LIN {X 0,Y 256.306,Z 543.369,A -85,B 0,C 180,E1 -18708.933,E2 -18708.933} C_VEL
LIN {X 0,Y 256.535,Z 543.34,A -85,B 0,C 180,E1 -18712.126,E2 -18712.126} C_VEL
LIN {X 0,Y 256.709,Z 543.322,A -85,B 0,C 180,E1 -18718.431,E2 -18718.431} C_VEL
LIN {X 0,Y 256.709,Z 543.317,A -85,B 0,C 180,E1 -18721.568,E2 -18721.568} C_VEL
LIN {X 0,Y 256.532,Z 543.34,A -85,B 0,C 180,E1 -18727.873,E2 -18727.873} C_VEL
LIN {X 0,Y 256.304,Z 543.369,A -85,B 0,C 180,E1 -18731.066,E2 -18731.066} C_VEL
LIN {X 0,Y 256.289,Z 543.37,A -85,B 0,C 180,E1 -18735.915,E2 -18735.915} C_VEL
LIN {X 0,Y 256.155,Z 543.39,A -85,B 0,C 180,E1 -18740.925,E2 -18740.925} C_VEL
LIN {X 0,Y 256.166,Z 543.386,A -85,B 0,C 180,E1 -18745.13,E2 -18745.13} C_VEL
LIN {X 0,Y 256.134,Z 543.388,A -85,B 0,C 180,E1 -18747.754,E2 -18747.754} C_VEL
LIN {X 0,Y 255.867,Z 543.426,A -85,B 0,C 180,E1 -18748.632,E2 -18748.632} C_VEL
LIN {X 0,Y 254.547,Z 543.595,A -85,B 0,C 180,E1 -18749.928,E2 -18749.928} C_VEL
LIN {X 0,Y 250.177,Z 544.136,A -85,B 0,C 180,E1 -18752.946,E2 -18752.946} C_VEL
LIN {X 0,Y 249.117,Z 544.265,A -85,B 0,C 180,E1 -18754.298,E2 -18754.298} C_VEL
LIN {X 0,Y 249.035,Z 544.274,A -85,B 0,C 180,E1 -18754.757,E2 -18754.757} C_VEL
LIN {X 0,Y 249.021,Z 544.276,A -85,B 0,C 180,E1 -18758.381,E2 -18758.381} C_VEL
LIN {X 0,Y 249.008,Z 544.281,A -85,B 0,C 180,E1 -18762.793,E2 -18762.793} C_VEL
LIN {X 0,Y 249.015,Z 544.278,A -85,B 0,C 180,E1 -18767.364,E2 -18767.364} C_VEL
LIN {X 0,Y 249.084,Z 544.269,A -85,B 0,C 180,E1 -18772.188,E2 -18772.188} C_VEL
LIN {X 0,Y 249.237,Z 544.478,A -85,B 0,C 180,E1 -18773.377,E2 -18773.377} C_VEL
LIN {X 0,Y 251.469,Z 555.944,A -85,B 0,C 180,E1 -18777.927,E2 -18777.927} C_VEL
LIN {X 0,Y 252.35,Z 561.158,A -85,B 0,C 180,E1 -18779.914,E2 -18779.914} C_VEL
LIN {X 0,Y 250.485,Z 573.384,A -85,B 0,C 180,E1 -18784.422,E2 -18784.422} C_VEL
LIN {X 0,Y 249.648,Z 580.162,A -85,B 0,C 180,E1 -18786.831,E2 -18786.831} C_VEL
LIN {X 0,Y 249.979,Z 590.6,A -85,B 0,C 180,E1 -18787.367,E2 -18787.367} C_VEL
LIN {X 0,Y 253.841,Z 654.438,A -85,B 0,C 180,E1 -18790.307,E2 -18790.307} C_VEL
LIN {X 0,Y 253.269,Z 669.393,A -85,B 0,C 180,E1 -18791.024,E2 -18791.024} C_VEL
LIN {X 0,Y 252.559,Z 681.968,A -85,B 0,C 180,E1 -18791.967,E2 -18791.967} C_VEL
LIN {X 0,Y 251.556,Z 693.327,A -85,B 0,C 180,E1 -18793.151,E2 -18793.151} C_VEL
LIN {X 0,Y 250.486,Z 703.576,A -85,B 0,C 180,E1 -18794.541,E2 -18794.541} C_VEL
LIN {X 0,Y 249.573,Z 714,A -85,B 0,C 180,E1 -18796.359,E2 -18796.359} C_VEL
LIN {X 0,Y 248.841,Z 722.24,A -85,B 0,C 180,E1 -18798.185,E2 -18798.185} C_VEL
LIN {X 0,Y 248.424,Z 729.674,A -85,B 0,C 180,E1 -18800.227,E2 -18800.227} C_VEL
LIN {X 0,Y 248.37,Z 736.358,A -85,B 0,C 180,E1 -18802.588,E2 -18802.588} C_VEL
LIN {X 0,Y 248.68,Z 741.797,A -85,B 0,C 180,E1 -18805.136,E2 -18805.136} C_VEL
LIN {X 0,Y 248.915,Z 744.383,A -85,B 0,C 180,E1 -18806.763,E2 -18806.763} C_VEL
LIN {X 0,Y 249.202,Z 746.318,A -85,B 0,C 180,E1 -18808.384,E2 -18808.384} C_VEL
LIN {X 0,Y 249.471,Z 747.677,A -85,B 0,C 180,E1 -18810,E2 -18810} C_VEL
LIN {X 0,Y 248.906,Z 748.281,A -85,B 0,C 180,E1 -18811.618,E2 -18811.618} C_VEL
LIN {X 0,Y 248.421,Z 748.396,A -85,B 0,C 180,E1 -18813.243,E2 -18813.243} C_VEL
LIN {X 0,Y 248.095,Z 747.972,A -85,B 0,C 180,E1 -18814.875,E2 -18814.875} C_VEL
LIN {X 0,Y 247.721,Z 746.838,A -85,B 0,C 180,E1 -18816.801,E2 -18816.801} C_VEL
LIN {X 0,Y 247.793,Z 743.709,A -85,B 0,C 180,E1 -18819.798,E2 -18819.798} C_VEL
LIN {X 0,Y 248.37,Z 739.868,A -85,B 0,C 180,E1 -18822.252,E2 -18822.252} C_VEL
LIN {X 0,Y 249.688,Z 734.737,A -85,B 0,C 180,E1 -18824.674,E2 -18824.674} C_VEL
LIN {X 0,Y 251.68,Z 728.243,A -85,B 0,C 180,E1 -18827.049,E2 -18827.049} C_VEL
LIN {X 0,Y 254.188,Z 720.034,A -85,B 0,C 180,E1 -18829.377,E2 -18829.377} C_VEL
LIN {X 0,Y 256.882,Z 711.584,A -85,B 0,C 180,E1 -18831.253,E2 -18831.253} C_VEL
LIN {X 0,Y 260.07,Z 700.565,A -85,B 0,C 180,E1 -18833.167,E2 -18833.167} C_VEL
LIN {X 0,Y 263.063,Z 689.343,A -85,B 0,C 180,E1 -18834.672,E2 -18834.672} C_VEL
LIN {X 0,Y 265.709,Z 677.727,A -85,B 0,C 180,E1 -18835.875,E2 -18835.875} C_VEL
LIN {X 0,Y 268.145,Z 664.605,A -85,B 0,C 180,E1 -18836.878,E2 -18836.878} C_VEL
LIN {X 0,Y 269.269,Z 654.548,A -85,B 0,C 180,E1 -18837.488,E2 -18837.488} C_VEL
LIN {X 0,Y 269.475,Z 635.451,A -85,B 0,C 180,E1 -18838.521,E2 -18838.521} C_VEL
LIN {X 0,Y 268.714,Z 621.119,A -85,B 0,C 180,E1 -18839.462,E2 -18839.462} C_VEL
LIN {X 0,Y 267.255,Z 606.263,A -85,B 0,C 180,E1 -18840.615,E2 -18840.615} C_VEL
LIN {X 0,Y 264.831,Z 589.544,A -85,B 0,C 180,E1 -18842.184,E2 -18842.184} C_VEL
LIN {X 0,Y 262.41,Z 576.84,A -85,B 0,C 180,E1 -18843.625,E2 -18843.625} C_VEL
LIN {X 0,Y 261.184,Z 573.597,A -85,B 0,C 180,E1 -18844.174,E2 -18844.174} C_VEL
LIN {X 0,Y 258.293,Z 566.656,A -85,B 0,C 180,E1 -18845.538,E2 -18845.538} C_VEL
LIN {X 0,Y 255.142,Z 559.582,A -85,B 0,C 180,E1 -18847.115,E2 -18847.115} C_VEL
LIN {X 0,Y 250.945,Z 551.351,A -85,B 0,C 180,E1 -18849.458,E2 -18849.458} C_VEL
LIN {X 0,Y 250.156,Z 548.87,A -85,B 0,C 180,E1 -18850.252,E2 -18850.252} C_VEL
LIN {X 0,Y 249.028,Z 544.337,A -85,B 0,C 180,E1 -18852.933,E2 -18852.933} C_VEL
LIN {X 0,Y 249.077,Z 544.264,A -85,B 0,C 180,E1 -18857.376,E2 -18857.376} C_VEL
LIN {X 0,Y 249.049,Z 544.268,A -85,B 0,C 180,E1 -18861.624,E2 -18861.624} C_VEL
LIN {X 0,Y 249.057,Z 544.274,A -85,B 0,C 180,E1 -18865.642,E2 -18865.642} C_VEL
LIN {X 0,Y 249.043,Z 544.273,A -85,B 0,C 180,E1 -18869.472,E2 -18869.472} C_VEL
LIN {X 0,Y 249.067,Z 544.266,A -85,B 0,C 180,E1 -18873.162,E2 -18873.162} C_VEL
LIN {X 0,Y 249.075,Z 544.264,A -85,B 0,C 180,E1 -18876.733,E2 -18876.733} C_VEL
LIN {X 0,Y 249.163,Z 544.496,A -85,B 0,C 180,E1 -18880.216,E2 -18880.216} C_VEL
LIN {X 0,Y 249.359,Z 545.297,A -85,B 0,C 180,E1 -18880.704,E2 -18880.704} C_VEL
LIN {X 0,Y 250.79,Z 548.019,A -85,B 0,C 180,E1 -18881.619,E2 -18881.619} C_VEL
LIN {X 0,Y 253.524,Z 550.284,A -85,B 0,C 180,E1 -18882.917,E2 -18882.917} C_VEL
LIN {X 0,Y 255.381,Z 553.409,A -85,B 0,C 180,E1 -18883.866,E2 -18883.866} C_VEL
LIN {X 0,Y 257.263,Z 555.416,A -85,B 0,C 180,E1 -18884.655,E2 -18884.655} C_VEL
LIN {X 0,Y 259.711,Z 558.996,A -85,B 0,C 180,E1 -18885.705,E2 -18885.705} C_VEL
LIN {X 0,Y 261.019,Z 560.888,A -85,B 0,C 180,E1 -18886.224,E2 -18886.224} C_VEL
LIN {X 0,Y 263.946,Z 565.055,A -85,B 0,C 180,E1 -18887.308,E2 -18887.308} C_VEL
LIN {X 0,Y 268.158,Z 571.387,A -85,B 0,C 180,E1 -18888.768,E2 -18888.768} C_VEL
LIN {X 0,Y 273.128,Z 580.703,A -85,B 0,C 180,E1 -18890.404,E2 -18890.404} C_VEL
LIN {X 0,Y 275.101,Z 584.615,A -85,B 0,C 180,E1 -18891.011,E2 -18891.011} C_VEL
LIN {X 0,Y 274.575,Z 597.999,A -85,B 0,C 180,E1 -18891.692,E2 -18891.692} C_VEL
LIN {X 0,Y 273.552,Z 610.337,A -85,B 0,C 180,E1 -18892.62,E2 -18892.62} C_VEL
LIN {X 0,Y 272.024,Z 621.323,A -85,B 0,C 180,E1 -18893.709,E2 -18893.709} C_VEL
LIN {X 0,Y 269.941,Z 632.521,A -85,B 0,C 180,E1 -18895.147,E2 -18895.147} C_VEL
LIN {X 0,Y 267.448,Z 643.158,A -85,B 0,C 180,E1 -18896.902,E2 -18896.902} C_VEL
LIN {X 0,Y 264.894,Z 652.456,A -85,B 0,C 180,E1 -18898.86,E2 -18898.86} C_VEL
LIN {X 0,Y 262.485,Z 659.657,A -85,B 0,C 180,E1 -18900.768,E2 -18900.768} C_VEL
LIN {X 0,Y 259.841,Z 666.594,A -85,B 0,C 180,E1 -18903.101,E2 -18903.101} C_VEL
LIN {X 0,Y 257.472,Z 671.988,A -85,B 0,C 180,E1 -18905.483,E2 -18905.483} C_VEL
LIN {X 0,Y 255.404,Z 676.066,A -85,B 0,C 180,E1 -18907.909,E2 -18907.909} C_VEL
LIN {X 0,Y 254.239,Z 678.115,A -85,B 0,C 180,E1 -18909.548,E2 -18909.548} C_VEL
LIN {X 0,Y 253.132,Z 679.649,A -85,B 0,C 180,E1 -18911.207,E2 -18911.207} C_VEL
LIN {X 0,Y 252.188,Z 680.696,A -85,B 0,C 180,E1 -18912.883,E2 -18912.883} C_VEL
LIN {X 0,Y 251.38,Z 681.261,A -85,B 0,C 180,E1 -18914.574,E2 -18914.574} C_VEL
LIN {X 0,Y 250.368,Z 681.117,A -85,B 0,C 180,E1 -18917.374,E2 -18917.374} C_VEL
LIN {X 0,Y 249.802,Z 680.003,A -85,B 0,C 180,E1 -18919.732,E2 -18919.732} C_VEL
LIN {X 0,Y 249.521,Z 678.439,A -85,B 0,C 180,E1 -18921.65,E2 -18921.65} C_VEL
LIN {X 0,Y 249.424,Z 675.466,A -85,B 0,C 180,E1 -18924.115,E2 -18924.115} C_VEL
LIN {X 0,Y 249.624,Z 671.003,A -85,B 0,C 180,E1 -18926.775,E2 -18926.775} C_VEL
LIN {X 0,Y 250.049,Z 665.232,A -85,B 0,C 180,E1 -18929.392,E2 -18929.392} C_VEL
LIN {X 0,Y 250.666,Z 658.689,A -85,B 0,C 180,E1 -18931.716,E2 -18931.716} C_VEL
LIN {X 0,Y 251.462,Z 650.773,A -85,B 0,C 180,E1 -18933.986,E2 -18933.986} C_VEL
LIN {X 0,Y 252.442,Z 641.376,A -85,B 0,C 180,E1 -18936.163,E2 -18936.163} C_VEL
LIN {X 0,Y 253.428,Z 630.912,A -85,B 0,C 180,E1 -18938.1,E2 -18938.1} C_VEL
LIN {X 0,Y 254.358,Z 620.06,A -85,B 0,C 180,E1 -18939.715,E2 -18939.715} C_VEL
LIN {X 0,Y 255.201,Z 608.035,A -85,B 0,C 180,E1 -18941.11,E2 -18941.11} C_VEL
LIN {X 0,Y 255.904,Z 595.234,A -85,B 0,C 180,E1 -18942.227,E2 -18942.227} C_VEL
LIN {X 0,Y 256.258,Z 581.462,A -85,B 0,C 180,E1 -18943.061,E2 -18943.061} C_VEL
LIN {X 0,Y 256.325,Z 567.498,A -85,B 0,C 180,E1 -18943.614,E2 -18943.614} C_VEL
LIN {X 0,Y 249.318,Z 545.365,A -85,B 0,C 180,E1 -18944.845,E2 -18944.845} C_VEL
LIN {X 0,Y 249.078,Z 544.391,A -85,B 0,C 180,E1 -18945.14,E2 -18945.14} C_VEL
LIN {X 0,Y 249.08,Z 544.273,A -85,B 0,C 180,E1 -18949.627,E2 -18949.627} C_VEL
LIN {X 0,Y 249.076,Z 544.272,A -85,B 0,C 180,E1 -18953.664,E2 -18953.664} C_VEL
LIN {X 0,Y 249.041,Z 544.276,A -85,B 0,C 180,E1 -18957.846,E2 -18957.846} C_VEL
LIN {X 0,Y 249.099,Z 544.27,A -85,B 0,C 180,E1 -18961.339,E2 -18961.339} C_VEL
LIN {X 0,Y 249.154,Z 544.26,A -85,B 0,C 180,E1 -18964.97,E2 -18964.97} C_VEL
LIN {X 0,Y 249.097,Z 544.266,A -85,B 0,C 180,E1 -18968.603,E2 -18968.603} C_VEL
LIN {X 0,Y 249.199,Z 544.255,A -85,B 0,C 180,E1 -18973.619,E2 -18973.619} C_VEL
LIN {X 0,Y 249.247,Z 544.248,A -85,B 0,C 180,E1 -18978.617,E2 -18978.617} C_VEL
LIN {X 0,Y 249.443,Z 544.224,A -85,B 0,C 180,E1 -18981.902,E2 -18981.902} C_VEL
LIN {X 0,Y 249.291,Z 544.243,A -85,B 0,C 180,E1 -18985.149,E2 -18985.149} C_VEL
LIN {X 0,Y 249.679,Z 544.194,A -85,B 0,C 180,E1 -18988.387,E2 -18988.387} C_VEL
LIN {X 0,Y 249.679,Z 544.195,A -85,B 0,C 180,E1 -18991.613,E2 -18991.613} C_VEL
LIN {X 0,Y 249.441,Z 544.224,A -85,B 0,C 180,E1 -18996.471,E2 -18996.471} C_VEL
LIN {X 0,Y 249.347,Z 544.237,A -85,B 0,C 180,E1 -18999.736,E2 -18999.736} C_VEL
LIN {X 0,Y 249.21,Z 544.253,A -85,B 0,C 180,E1 -19004.703,E2 -19004.703} C_VEL
LIN {X 0,Y 249.143,Z 544.261,A -85,B 0,C 180,E1 -19008.077,E2 -19008.077} C_VEL
LIN {X 0,Y 249.087,Z 544.268,A -85,B 0,C 180,E1 -19011.518,E2 -19011.518} C_VEL
LIN {X 0,Y 249.12,Z 544.265,A -85,B 0,C 180,E1 -19015.475,E2 -19015.475} C_VEL
LIN {X 0,Y 249.075,Z 544.267,A -85,B 0,C 180,E1 -19018.988,E2 -19018.988} C_VEL
LIN {X 0,Y 249.038,Z 544.275,A -85,B 0,C 180,E1 -19022.424,E2 -19022.424} C_VEL
LIN {X 0,Y 249.077,Z 544.268,A -85,B 0,C 180,E1 -19026.337,E2 -19026.337} C_VEL
LIN {X 0,Y 249.079,Z 544.271,A -85,B 0,C 180,E1 -19030.463,E2 -19030.463} C_VEL
LIN {X 0,Y 249.02,Z 544.274,A -85,B 0,C 180,E1 -19034.874,E2 -19034.874} C_VEL
LIN {X 0,Y 249.024,Z 544.274,A -85,B 0,C 180,E1 -19037.364,E2 -19037.364} C_VEL
LIN {X 0,Y 249.047,Z 544.276,A -85,B 0,C 180,E1 -19042.198,E2 -19042.198} C_VEL
LIN {X 0,Y 249.057,Z 544.27,A -85,B 0,C 180,E1 -19045.641,E2 -19045.641} C_VEL
LIN {X 0,Y 249.049,Z 544.273,A -85,B 0,C 180,E1 -19049.472,E2 -19049.472} C_VEL
LIN {X 0,Y 249.07,Z 544.267,A -85,B 0,C 180,E1 -19053.161,E2 -19053.161} C_VEL
LIN {X 0,Y 249.082,Z 544.27,A -85,B 0,C 180,E1 -19056.732,E2 -19056.732} C_VEL
LIN {X 0,Y 249.127,Z 544.266,A -85,B 0,C 180,E1 -19060.212,E2 -19060.212} C_VEL
LIN {X 0,Y 249.239,Z 544.247,A -85,B 0,C 180,E1 -19063.621,E2 -19063.621} C_VEL
LIN {X 0,Y 249.249,Z 544.25,A -85,B 0,C 180,E1 -19068.616,E2 -19068.616} C_VEL
LIN {X 0,Y 249.477,Z 544.217,A -85,B 0,C 180,E1 -19071.902,E2 -19071.902} C_VEL
LIN {X 0,Y 249.432,Z 544.227,A -85,B 0,C 180,E1 -19076.769,E2 -19076.769} C_VEL
LIN {X 0,Y 249.723,Z 544.188,A -85,B 0,C 180,E1 -19079.999,E2 -19079.999} C_VEL
LIN {X 0,Y 249.431,Z 544.225,A -85,B 0,C 180,E1 -19083.23,E2 -19083.23} C_VEL
LIN {X 0,Y 249.474,Z 544.22,A -85,B 0,C 180,E1 -19088.097,E2 -19088.097} C_VEL
LIN {X 0,Y 249.247,Z 544.247,A -85,B 0,C 180,E1 -19091.383,E2 -19091.383} C_VEL
LIN {X 0,Y 249.213,Z 544.255,A -85,B 0,C 180,E1 -19096.503,E2 -19096.503} C_VEL
LIN {X 0,Y 249.079,Z 544.269,A -85,B 0,C 180,E1 -19101.518,E2 -19101.518} C_VEL
LIN {X 0,Y 249.113,Z 544.263,A -85,B 0,C 180,E1 -19105.476,E2 -19105.476} C_VEL
LIN {X 0,Y 249.079,Z 544.271,A -85,B 0,C 180,E1 -19108.993,E2 -19108.993} C_VEL
LIN {X 0,Y 249.026,Z 544.277,A -85,B 0,C 180,E1 -19112.426,E2 -19112.426} C_VEL
LIN {X 0,Y 249.035,Z 544.274,A -85,B 0,C 180,E1 -19114.757,E2 -19114.757} C_VEL
LIN {X 0,Y 248.384,Z 544.355,A -85,B 0,C 180,E1 -19116.106,E2 -19116.106} C_VEL
LIN {X 0,Y 245.551,Z 544.714,A -85,B 0,C 180,E1 -19118.308,E2 -19118.308} C_VEL
LIN {X 0,Y 243.114,Z 545.018,A -85,B 0,C 180,E1 -19120.099,E2 -19120.099} C_VEL
LIN {X 0,Y 242.037,Z 545.148,A -85,B 0,C 180,E1 -19121.489,E2 -19121.489} C_VEL
LIN {X 0,Y 241.933,Z 545.158,A -85,B 0,C 180,E1 -19121.961,E2 -19121.961} C_VEL
LIN {X 0,Y 241.933,Z 545.161,A -85,B 0,C 180,E1 -19126.571,E2 -19126.571} C_VEL
LIN {X 0,Y 241.974,Z 545.155,A -85,B 0,C 180,E1 -19130.285,E2 -19130.285} C_VEL
LIN {X 0,Y 242.181,Z 545.268,A -85,B 0,C 180,E1 -19133.263,E2 -19133.263} C_VEL
LIN {X 0,Y 244.353,Z 556.428,A -85,B 0,C 180,E1 -19137.854,E2 -19137.854} C_VEL
LIN {X 0,Y 245.133,Z 560.149,A -85,B 0,C 180,E1 -19139.328,E2 -19139.328} C_VEL
LIN {X 0,Y 245.169,Z 562.117,A -85,B 0,C 180,E1 -19140.087,E2 -19140.087} C_VEL
LIN {X 0,Y 243.221,Z 574.405,A -85,B 0,C 180,E1 -19144.773,E2 -19144.773} C_VEL
LIN {X 0,Y 242.685,Z 578.872,A -85,B 0,C 180,E1 -19146.403,E2 -19146.403} C_VEL
LIN {X 0,Y 243.22,Z 594.089,A -85,B 0,C 180,E1 -19147.176,E2 -19147.176} C_VEL
LIN {X 0,Y 246.829,Z 654.667,A -85,B 0,C 180,E1 -19150.066,E2 -19150.066} C_VEL
LIN {X 0,Y 246.25,Z 669.144,A -85,B 0,C 180,E1 -19150.808,E2 -19150.808} C_VEL
LIN {X 0,Y 245.536,Z 681.208,A -85,B 0,C 180,E1 -19151.756,E2 -19151.756} C_VEL
LIN {X 0,Y 244.635,Z 691.628,A -85,B 0,C 180,E1 -19152.875,E2 -19152.875} C_VEL
LIN {X 0,Y 243.5,Z 701.966,A -85,B 0,C 180,E1 -19154.301,E2 -19154.301} C_VEL
LIN {X 0,Y 242.595,Z 712.471,A -85,B 0,C 180,E1 -19156.173,E2 -19156.173} C_VEL
LIN {X 0,Y 241.906,Z 719.97,A -85,B 0,C 180,E1 -19157.841,E2 -19157.841} C_VEL
LIN {X 0,Y 241.44,Z 727.586,A -85,B 0,C 180,E1 -19159.942,E2 -19159.942} C_VEL
LIN {X 0,Y 241.353,Z 733.346,A -85,B 0,C 180,E1 -19161.909,E2 -19161.909} C_VEL
LIN {X 0,Y 241.55,Z 738.574,A -85,B 0,C 180,E1 -19164.155,E2 -19164.155} C_VEL
LIN {X 0,Y 241.929,Z 742.872,A -85,B 0,C 180,E1 -19166.669,E2 -19166.669} C_VEL
LIN {X 0,Y 242.198,Z 744.937,A -85,B 0,C 180,E1 -19168.337,E2 -19168.337} C_VEL
LIN {X 0,Y 242.487,Z 746.367,A -85,B 0,C 180,E1 -19170,E2 -19170} C_VEL
LIN {X 0,Y 241.879,Z 747.084,A -85,B 0,C 180,E1 -19171.665,E2 -19171.665} C_VEL
LIN {X 0,Y 241.369,Z 747.254,A -85,B 0,C 180,E1 -19173.338,E2 -19173.338} C_VEL
LIN {X 0,Y 241.024,Z 746.946,A -85,B 0,C 180,E1 -19175.018,E2 -19175.018} C_VEL
LIN {X 0,Y 240.682,Z 745.98,A -85,B 0,C 180,E1 -19176.878,E2 -19176.878} C_VEL
LIN {X 0,Y 240.621,Z 744.785,A -85,B 0,C 180,E1 -19178.397,E2 -19178.397} C_VEL
LIN {X 0,Y 240.885,Z 741.864,A -85,B 0,C 180,E1 -19180.932,E2 -19180.932} C_VEL
LIN {X 0,Y 241.745,Z 737.782,A -85,B 0,C 180,E1 -19183.448,E2 -19183.448} C_VEL
LIN {X 0,Y 243.443,Z 732.479,A -85,B 0,C 180,E1 -19185.917,E2 -19185.917} C_VEL
LIN {X 0,Y 245.657,Z 725.699,A -85,B 0,C 180,E1 -19188.342,E2 -19188.342} C_VEL
LIN {X 0,Y 248.57,Z 717.168,A -85,B 0,C 180,E1 -19190.696,E2 -19190.696} C_VEL
LIN {X 0,Y 251.557,Z 708.396,A -85,B 0,C 180,E1 -19192.59,E2 -19192.59} C_VEL
LIN {X 0,Y 254.501,Z 698.752,A -85,B 0,C 180,E1 -19194.263,E2 -19194.263} C_VEL
LIN {X 0,Y 257.45,Z 688.25,A -85,B 0,C 180,E1 -19195.68,E2 -19195.68} C_VEL
LIN {X 0,Y 260.219,Z 676.714,A -85,B 0,C 180,E1 -19196.896,E2 -19196.896} C_VEL
LIN {X 0,Y 262.767,Z 663.786,A -85,B 0,C 180,E1 -19197.908,E2 -19197.908} C_VEL
LIN {X 0,Y 263.92,Z 654.338,A -85,B 0,C 180,E1 -19198.522,E2 -19198.522} C_VEL
LIN {X 0,Y 264.358,Z 637.592,A -85,B 0,C 180,E1 -19199.478,E2 -19199.478} C_VEL
LIN {X 0,Y 263.68,Z 622.935,A -85,B 0,C 180,E1 -19200.463,E2 -19200.463} C_VEL
LIN {X 0,Y 262.372,Z 608.127,A -85,B 0,C 180,E1 -19201.661,E2 -19201.661} C_VEL
LIN {X 0,Y 260.248,Z 592.266,A -85,B 0,C 180,E1 -19203.211,E2 -19203.211} C_VEL
LIN {X 0,Y 258.202,Z 580.621,A -85,B 0,C 180,E1 -19204.581,E2 -19204.581} C_VEL
LIN {X 0,Y 256.941,Z 577.281,A -85,B 0,C 180,E1 -19205.209,E2 -19205.209} C_VEL
LIN {X 0,Y 254.616,Z 571.474,A -85,B 0,C 180,E1 -19206.382,E2 -19206.382} C_VEL
LIN {X 0,Y 251.313,Z 563.79,A -85,B 0,C 180,E1 -19208.213,E2 -19208.213} C_VEL
LIN {X 0,Y 248.064,Z 557.057,A -85,B 0,C 180,E1 -19210.177,E2 -19210.177} C_VEL
LIN {X 0,Y 246.842,Z 554.324,A -85,B 0,C 180,E1 -19211.018,E2 -19211.018} C_VEL
LIN {X 0,Y 243.727,Z 548.974,A -85,B 0,C 180,E1 -19213.273,E2 -19213.273} C_VEL
LIN {X 0,Y 242.319,Z 546.623,A -85,B 0,C 180,E1 -19214.505,E2 -19214.505} C_VEL
LIN {X 0,Y 242.053,Z 545.556,A -85,B 0,C 180,E1 -19215.092,E2 -19215.092} C_VEL
LIN {X 0,Y 241.997,Z 545.153,A -85,B 0,C 180,E1 -19216.554,E2 -19216.554} C_VEL
LIN {X 0,Y 242.006,Z 545.146,A -85,B 0,C 180,E1 -19220.291,E2 -19220.291} C_VEL
LIN {X 0,Y 242.032,Z 545.14,A -85,B 0,C 180,E1 -19224.497,E2 -19224.497} C_VEL
LIN {X 0,Y 241.97,Z 545.152,A -85,B 0,C 180,E1 -19228.48,E2 -19228.48} C_VEL
LIN {X 0,Y 241.998,Z 545.154,A -85,B 0,C 180,E1 -19232.312,E2 -19232.312} C_VEL
LIN {X 0,Y 242.052,Z 545.284,A -85,B 0,C 180,E1 -19236.016,E2 -19236.016} C_VEL
LIN {X 0,Y 242.246,Z 546.171,A -85,B 0,C 180,E1 -19236.847,E2 -19236.847} C_VEL
LIN {X 0,Y 243.438,Z 548.608,A -85,B 0,C 180,E1 -19237.957,E2 -19237.957} C_VEL
LIN {X 0,Y 245.997,Z 550.658,A -85,B 0,C 180,E1 -19239.591,E2 -19239.591} C_VEL
LIN {X 0,Y 246.798,Z 551.349,A -85,B 0,C 180,E1 -19240.067,E2 -19240.067} C_VEL
LIN {X 0,Y 248.354,Z 554.312,A -85,B 0,C 180,E1 -19241.115,E2 -19241.115} C_VEL
LIN {X 0,Y 250.926,Z 556.718,A -85,B 0,C 180,E1 -19242.404,E2 -19242.404} C_VEL
LIN {X 0,Y 253.029,Z 559.959,A -85,B 0,C 180,E1 -19243.501,E2 -19243.501} C_VEL
LIN {X 0,Y 254.429,Z 561.588,A -85,B 0,C 180,E1 -19244.12,E2 -19244.12} C_VEL
LIN {X 0,Y 257.935,Z 566.768,A -85,B 0,C 180,E1 -19245.654,E2 -19245.654} C_VEL
LIN {X 0,Y 260.811,Z 571.029,A -85,B 0,C 180,E1 -19246.782,E2 -19246.782} C_VEL
LIN {X 0,Y 264.596,Z 577.005,A -85,B 0,C 180,E1 -19248.182,E2 -19248.182} C_VEL
LIN {X 0,Y 268.645,Z 584.636,A -85,B 0,C 180,E1 -19249.582,E2 -19249.582} C_VEL
LIN {X 0,Y 270.091,Z 587.626,A -85,B 0,C 180,E1 -19250.07,E2 -19250.07} C_VEL
LIN {X 0,Y 269.417,Z 600.249,A -85,B 0,C 180,E1 -19250.754,E2 -19250.754} C_VEL
LIN {X 0,Y 268.194,Z 612.764,A -85,B 0,C 180,E1 -19251.738,E2 -19251.738} C_VEL
LIN {X 0,Y 266.361,Z 624.735,A -85,B 0,C 180,E1 -19252.991,E2 -19252.991} C_VEL
LIN {X 0,Y 264.409,Z 634.383,A -85,B 0,C 180,E1 -19254.28,E2 -19254.28} C_VEL
LIN {X 0,Y 262.221,Z 643.27,A -85,B 0,C 180,E1 -19255.768,E2 -19255.768} C_VEL
LIN {X 0,Y 259.538,Z 652.374,A -85,B 0,C 180,E1 -19257.672,E2 -19257.672} C_VEL
LIN {X 0,Y 256.935,Z 659.845,A -85,B 0,C 180,E1 -19259.609,E2 -19259.609} C_VEL
LIN {X 0,Y 254.545,Z 665.938,A -85,B 0,C 180,E1 -19261.583,E2 -19261.583} C_VEL
LIN {X 0,Y 251.942,Z 671.729,A -85,B 0,C 180,E1 -19264,E2 -19264} C_VEL
LIN {X 0,Y 249.629,Z 676.167,A -85,B 0,C 180,E1 -19266.467,E2 -19266.467} C_VEL
LIN {X 0,Y 248.254,Z 678.436,A -85,B 0,C 180,E1 -19268.138,E2 -19268.138} C_VEL
LIN {X 0,Y 247.016,Z 680.18,A -85,B 0,C 180,E1 -19269.83,E2 -19269.83} C_VEL
LIN {X 0,Y 245.917,Z 681.462,A -85,B 0,C 180,E1 -19271.541,E2 -19271.541} C_VEL
LIN {X 0,Y 244.975,Z 682.215,A -85,B 0,C 180,E1 -19273.269,E2 -19273.269} C_VEL
LIN {X 0,Y 244.181,Z 682.521,A -85,B 0,C 180,E1 -19275.014,E2 -19275.014} C_VEL
LIN {X 0,Y 243.283,Z 682.064,A -85,B 0,C 180,E1 -19277.582,E2 -19277.582} C_VEL
LIN {X 0,Y 242.638,Z 680.415,A -85,B 0,C 180,E1 -19280.34,E2 -19280.34} C_VEL
LIN {X 0,Y 242.359,Z 677.64,A -85,B 0,C 180,E1 -19283.047,E2 -19283.047} C_VEL
LIN {X 0,Y 242.487,Z 673.147,A -85,B 0,C 180,E1 -19286.045,E2 -19286.045} C_VEL
LIN {X 0,Y 242.871,Z 667.018,A -85,B 0,C 180,E1 -19288.993,E2 -19288.993} C_VEL
LIN {X 0,Y 243.473,Z 660.892,A -85,B 0,C 180,E1 -19291.305,E2 -19291.305} C_VEL
LIN {X 0,Y 244.252,Z 653.107,A -85,B 0,C 180,E1 -19293.672,E2 -19293.672} C_VEL
LIN {X 0,Y 245.236,Z 643.667,A -85,B 0,C 180,E1 -19295.98,E2 -19295.98} C_VEL
LIN {X 0,Y 246.18,Z 634.123,A -85,B 0,C 180,E1 -19297.865,E2 -19297.865} C_VEL
LIN {X 0,Y 247.28,Z 622.008,A -85,B 0,C 180,E1 -19299.769,E2 -19299.769} C_VEL
LIN {X 0,Y 248.08,Z 610.304,A -85,B 0,C 180,E1 -19301.199,E2 -19301.199} C_VEL
LIN {X 0,Y 248.864,Z 597.366,A -85,B 0,C 180,E1 -19302.396,E2 -19302.396} C_VEL
LIN {X 0,Y 249.271,Z 583.964,A -85,B 0,C 180,E1 -19303.262,E2 -19303.262} C_VEL
LIN {X 0,Y 249.363,Z 568.727,A -85,B 0,C 180,E1 -19303.911,E2 -19303.911} C_VEL
LIN {X 0,Y 242.192,Z 545.985,A -85,B 0,C 180,E1 -19305.241,E2 -19305.241} C_VEL
LIN {X 0,Y 242.035,Z 545.237,A -85,B 0,C 180,E1 -19305.533,E2 -19305.533} C_VEL
LIN {X 0,Y 242.008,Z 545.151,A -85,B 0,C 180,E1 -19310.292,E2 -19310.292} C_VEL
LIN {X 0,Y 242.038,Z 545.146,A -85,B 0,C 180,E1 -19314.499,E2 -19314.499} C_VEL
LIN {X 0,Y 241.978,Z 545.154,A -85,B 0,C 180,E1 -19318.481,E2 -19318.481} C_VEL
LIN {X 0,Y 242.011,Z 545.149,A -85,B 0,C 180,E1 -19322.314,E2 -19322.314} C_VEL
LIN {X 0,Y 242.059,Z 545.143,A -85,B 0,C 180,E1 -19326.017,E2 -19326.017} C_VEL
LIN {X 0,Y 242.032,Z 545.151,A -85,B 0,C 180,E1 -19329.608,E2 -19329.608} C_VEL
LIN {X 0,Y 242.119,Z 545.136,A -85,B 0,C 180,E1 -19333.317,E2 -19333.317} C_VEL
LIN {X 0,Y 242.158,Z 545.131,A -85,B 0,C 180,E1 -19336.575,E2 -19336.575} C_VEL
LIN {X 0,Y 242.392,Z 545.103,A -85,B 0,C 180,E1 -19341.665,E2 -19341.665} C_VEL
LIN {X 0,Y 242.251,Z 545.119,A -85,B 0,C 180,E1 -19345.007,E2 -19345.007} C_VEL
LIN {X 0,Y 242.64,Z 545.071,A -85,B 0,C 180,E1 -19348.34,E2 -19348.34} C_VEL
LIN {X 0,Y 242.64,Z 545.072,A -85,B 0,C 180,E1 -19351.66,E2 -19351.66} C_VEL
LIN {X 0,Y 242.412,Z 545.099,A -85,B 0,C 180,E1 -19356.659,E2 -19356.659} C_VEL
LIN {X 0,Y 242.271,Z 545.117,A -85,B 0,C 180,E1 -19360.023,E2 -19360.023} C_VEL
LIN {X 0,Y 242.171,Z 545.13,A -85,B 0,C 180,E1 -19365.14,E2 -19365.14} C_VEL
LIN {X 0,Y 242.076,Z 545.138,A -85,B 0,C 180,E1 -19368.624,E2 -19368.624} C_VEL
LIN {X 0,Y 242.01,Z 545.152,A -85,B 0,C 180,E1 -19372.18,E2 -19372.18} C_VEL
LIN {X 0,Y 242.069,Z 545.145,A -85,B 0,C 180,E1 -19375.837,E2 -19375.837} C_VEL
LIN {X 0,Y 242.009,Z 545.149,A -85,B 0,C 180,E1 -19379.582,E2 -19379.582} C_VEL
LIN {X 0,Y 241.993,Z 545.152,A -85,B 0,C 180,E1 -19383.49,E2 -19383.49} C_VEL
LIN {X 0,Y 242.014,Z 545.147,A -85,B 0,C 180,E1 -19387.576,E2 -19387.576} C_VEL
LIN {X 0,Y 241.986,Z 545.156,A -85,B 0,C 180,E1 -19391.911,E2 -19391.911} C_VEL
LIN {X 0,Y 241.943,Z 545.158,A -85,B 0,C 180,E1 -19395.8,E2 -19395.8} C_VEL
LIN {X 0,Y 241.957,Z 545.159,A -85,B 0,C 180,E1 -19400.28,E2 -19400.28} C_VEL
LIN {X 0,Y 242.036,Z 545.146,A -85,B 0,C 180,E1 -19404.496,E2 -19404.496} C_VEL
LIN {X 0,Y 241.974,Z 545.156,A -85,B 0,C 180,E1 -19408.479,E2 -19408.479} C_VEL
LIN {X 0,Y 242.005,Z 545.151,A -85,B 0,C 180,E1 -19412.312,E2 -19412.312} C_VEL
LIN {X 0,Y 242.057,Z 545.145,A -85,B 0,C 180,E1 -19416.015,E2 -19416.015} C_VEL
LIN {X 0,Y 242.058,Z 545.143,A -85,B 0,C 180,E1 -19419.609,E2 -19419.609} C_VEL
LIN {X 0,Y 242.16,Z 545.128,A -85,B 0,C 180,E1 -19423.277,E2 -19423.277} C_VEL
LIN {X 0,Y 242.182,Z 545.132,A -85,B 0,C 180,E1 -19428.279,E2 -19428.279} C_VEL
LIN {X 0,Y 242.423,Z 545.095,A -85,B 0,C 180,E1 -19431.665,E2 -19431.665} C_VEL
LIN {X 0,Y 242.256,Z 545.119,A -85,B 0,C 180,E1 -19435.007,E2 -19435.007} C_VEL
LIN {X 0,Y 242.632,Z 545.075,A -85,B 0,C 180,E1 -19438.34,E2 -19438.34} C_VEL
LIN {X 0,Y 242.631,Z 545.07,A -85,B 0,C 180,E1 -19441.659,E2 -19441.659} C_VEL
LIN {X 0,Y 242.426,Z 545.1,A -85,B 0,C 180,E1 -19446.658,E2 -19446.658} C_VEL
LIN {X 0,Y 242.309,Z 545.11,A -85,B 0,C 180,E1 -19450.021,E2 -19450.021} C_VEL
LIN {X 0,Y 242.159,Z 545.131,A -85,B 0,C 180,E1 -19455.141,E2 -19455.141} C_VEL
LIN {X 0,Y 242.066,Z 545.143,A -85,B 0,C 180,E1 -19458.624,E2 -19458.624} C_VEL
LIN {X 0,Y 242.002,Z 545.151,A -85,B 0,C 180,E1 -19462.18,E2 -19462.18} C_VEL
LIN {X 0,Y 242.062,Z 545.141,A -85,B 0,C 180,E1 -19465.838,E2 -19465.838} C_VEL
LIN {X 0,Y 242.026,Z 545.147,A -85,B 0,C 180,E1 -19469.58,E2 -19469.58} C_VEL
LIN {X 0,Y 241.976,Z 545.153,A -85,B 0,C 180,E1 -19473.493,E2 -19473.493} C_VEL
LIN {X 0,Y 241.982,Z 545.152,A -85,B 0,C 180,E1 -19477.583,E2 -19477.583} C_VEL
LIN {X 0,Y 241.933,Z 545.158,A -85,B 0,C 180,E1 -19481.961,E2 -19481.961} C_VEL
LIN {X 0,Y 241.224,Z 545.249,A -85,B 0,C 180,E1 -19483.35,E2 -19483.35} C_VEL
LIN {X 0,Y 238.376,Z 545.603,A -85,B 0,C 180,E1 -19485.618,E2 -19485.618} C_VEL
LIN {X 0,Y 235.985,Z 545.904,A -85,B 0,C 180,E1 -19487.465,E2 -19487.465} C_VEL
LIN {X 0,Y 234.962,Z 546.031,A -85,B 0,C 180,E1 -19488.898,E2 -19488.898} C_VEL
LIN {X 0,Y 234.879,Z 546.038,A -85,B 0,C 180,E1 -19489.383,E2 -19489.383} C_VEL
LIN {X 0,Y 235.167,Z 546.231,A -85,B 0,C 180,E1 -19493.295,E2 -19493.295} C_VEL
LIN {X 0,Y 237.583,Z 558.486,A -85,B 0,C 180,E1 -19498.449,E2 -19498.449} C_VEL
LIN {X 0,Y 238.079,Z 562.024,A -85,B 0,C 180,E1 -19499.879,E2 -19499.879} C_VEL
LIN {X 0,Y 236.248,Z 573.593,A -85,B 0,C 180,E1 -19504.447,E2 -19504.447} C_VEL
LIN {X 0,Y 235.712,Z 577.668,A -85,B 0,C 180,E1 -19505.974,E2 -19505.974} C_VEL
LIN {X 0,Y 236.026,Z 589.638,A -85,B 0,C 180,E1 -19506.619,E2 -19506.619} C_VEL
LIN {X 0,Y 239.79,Z 655.024,A -85,B 0,C 180,E1 -19509.849,E2 -19509.849} C_VEL
LIN {X 0,Y 239.23,Z 668.34,A -85,B 0,C 180,E1 -19510.571,E2 -19510.571} C_VEL
LIN {X 0,Y 238.532,Z 680.173,A -85,B 0,C 180,E1 -19511.535,E2 -19511.535} C_VEL
LIN {X 0,Y 237.54,Z 691.399,A -85,B 0,C 180,E1 -19512.791,E2 -19512.791} C_VEL
LIN {X 0,Y 236.436,Z 701.555,A -85,B 0,C 180,E1 -19514.262,E2 -19514.262} C_VEL
LIN {X 0,Y 235.529,Z 711.937,A -85,B 0,C 180,E1 -19516.19,E2 -19516.19} C_VEL
LIN {X 0,Y 234.73,Z 720.96,A -85,B 0,C 180,E1 -19518.34,E2 -19518.34} C_VEL
LIN {X 0,Y 234.359,Z 728.2,A -85,B 0,C 180,E1 -19520.507,E2 -19520.507} C_VEL
LIN {X 0,Y 234.399,Z 734.985,A -85,B 0,C 180,E1 -19523.112,E2 -19523.112} C_VEL
LIN {X 0,Y 234.765,Z 740.016,A -85,B 0,C 180,E1 -19525.708,E2 -19525.708} C_VEL
LIN {X 0,Y 235.192,Z 743.518,A -85,B 0,C 180,E1 -19528.288,E2 -19528.288} C_VEL
LIN {X 0,Y 235.494,Z 745.044,A -85,B 0,C 180,E1 -19530,E2 -19530} C_VEL
LIN {X 0,Y 234.876,Z 745.841,A -85,B 0,C 180,E1 -19531.715,E2 -19531.715} C_VEL
LIN {X 0,Y 234.319,Z 746.098,A -85,B 0,C 180,E1 -19533.439,E2 -19533.439} C_VEL
LIN {X 0,Y 233.955,Z 745.868,A -85,B 0,C 180,E1 -19535.17,E2 -19535.17} C_VEL
LIN {X 0,Y 233.639,Z 745.109,A -85,B 0,C 180,E1 -19536.95,E2 -19536.95} C_VEL
LIN {X 0,Y 233.562,Z 743.896,A -85,B 0,C 180,E1 -19538.653,E2 -19538.653} C_VEL
LIN {X 0,Y 233.883,Z 741.167,A -85,B 0,C 180,E1 -19541.263,E2 -19541.263} C_VEL
LIN {X 0,Y 234.819,Z 737.308,A -85,B 0,C 180,E1 -19543.853,E2 -19543.853} C_VEL
LIN {X 0,Y 236.99,Z 731.204,A -85,B 0,C 180,E1 -19546.806,E2 -19546.806} C_VEL
LIN {X 0,Y 239.389,Z 724.455,A -85,B 0,C 180,E1 -19549.285,E2 -19549.285} C_VEL
LIN {X 0,Y 242.576,Z 716.009,A -85,B 0,C 180,E1 -19551.678,E2 -19551.678} C_VEL
LIN {X 0,Y 245.71,Z 707.254,A -85,B 0,C 180,E1 -19553.605,E2 -19553.605} C_VEL
LIN {X 0,Y 248.791,Z 697.68,A -85,B 0,C 180,E1 -19555.293,E2 -19555.293} C_VEL
LIN {X 0,Y 252.276,Z 685.855,A -85,B 0,C 180,E1 -19556.916,E2 -19556.916} C_VEL
LIN {X 0,Y 255.323,Z 674.109,A -85,B 0,C 180,E1 -19558.123,E2 -19558.123} C_VEL
LIN {X 0,Y 257.94,Z 660.949,A -85,B 0,C 180,E1 -19559.145,E2 -19559.145} C_VEL
LIN {X 0,Y 259.19,Z 647.069,A -85,B 0,C 180,E1 -19560.052,E2 -19560.052} C_VEL
LIN {X 0,Y 259.131,Z 630.772,A -85,B 0,C 180,E1 -19561.066,E2 -19561.066} C_VEL
LIN {X 0,Y 258.069,Z 614.467,A -85,B 0,C 180,E1 -19562.364,E2 -19562.364} C_VEL
LIN {X 0,Y 256.478,Z 599.883,A -85,B 0,C 180,E1 -19563.751,E2 -19563.751} C_VEL
LIN {X 0,Y 254.274,Z 584.858,A -85,B 0,C 180,E1 -19565.501,E2 -19565.501} C_VEL
LIN {X 0,Y 251.192,Z 576.579,A -85,B 0,C 180,E1 -19567.199,E2 -19567.199} C_VEL
LIN {X 0,Y 248.182,Z 569.163,A -85,B 0,C 180,E1 -19568.996,E2 -19568.996} C_VEL
LIN {X 0,Y 245.199,Z 562.509,A -85,B 0,C 180,E1 -19570.996,E2 -19570.996} C_VEL
LIN {X 0,Y 244.196,Z 560.182,A -85,B 0,C 180,E1 -19571.731,E2 -19571.731} C_VEL
LIN {X 0,Y 241.445,Z 555.212,A -85,B 0,C 180,E1 -19573.908,E2 -19573.908} C_VEL
LIN {X 0,Y 240.012,Z 552.511,A -85,B 0,C 180,E1 -19575.258,E2 -19575.258} C_VEL
LIN {X 0,Y 239.105,Z 551.67,A -85,B 0,C 180,E1 -19576.065,E2 -19576.065} C_VEL
LIN {X 0,Y 236.175,Z 549.214,A -85,B 0,C 180,E1 -19579.388,E2 -19579.388} C_VEL
LIN {X 0,Y 235.097,Z 546.709,A -85,B 0,C 180,E1 -19582.206,E2 -19582.206} C_VEL
LIN {X 0,Y 234.96,Z 546.229,A -85,B 0,C 180,E1 -19585.368,E2 -19585.368} C_VEL
LIN {X 0,Y 235.007,Z 546.474,A -85,B 0,C 180,E1 -19588.444,E2 -19588.444} C_VEL
LIN {X 0,Y 235.266,Z 547.4,A -85,B 0,C 180,E1 -19590.147,E2 -19590.147} C_VEL
LIN {X 0,Y 237.372,Z 550.487,A -85,B 0,C 180,E1 -19593.634,E2 -19593.634} C_VEL
LIN {X 0,Y 240.002,Z 552.224,A -85,B 0,C 180,E1 -19596.143,E2 -19596.143} C_VEL
LIN {X 0,Y 241.186,Z 554.783,A -85,B 0,C 180,E1 -19597.289,E2 -19597.289} C_VEL
LIN {X 0,Y 243.979,Z 557.324,A -85,B 0,C 180,E1 -19599.229,E2 -19599.229} C_VEL
LIN {X 0,Y 244.632,Z 558.236,A -85,B 0,C 180,E1 -19599.663,E2 -19599.663} C_VEL
LIN {X 0,Y 246.543,Z 561.258,A -85,B 0,C 180,E1 -19600.917,E2 -19600.917} C_VEL
LIN {X 0,Y 248.411,Z 563.092,A -85,B 0,C 180,E1 -19601.895,E2 -19601.895} C_VEL
LIN {X 0,Y 250.768,Z 566.513,A -85,B 0,C 180,E1 -19603.14,E2 -19603.14} C_VEL
LIN {X 0,Y 254.917,Z 572.624,A -85,B 0,C 180,E1 -19605.061,E2 -19605.061} C_VEL
LIN {X 0,Y 259.243,Z 579.282,A -85,B 0,C 180,E1 -19606.839,E2 -19606.839} C_VEL
LIN {X 0,Y 263.034,Z 586.245,A -85,B 0,C 180,E1 -19608.298,E2 -19608.298} C_VEL
LIN {X 0,Y 265.136,Z 590.652,A -85,B 0,C 180,E1 -19609.071,E2 -19609.071} C_VEL
LIN {X 0,Y 264.375,Z 603.512,A -85,B 0,C 180,E1 -19609.833,E2 -19609.833} C_VEL
LIN {X 0,Y 263.043,Z 614.992,A -85,B 0,C 180,E1 -19610.776,E2 -19610.776} C_VEL
LIN {X 0,Y 261.044,Z 626.838,A -85,B 0,C 180,E1 -19612.07,E2 -19612.07} C_VEL
LIN {X 0,Y 258.685,Z 637.369,A -85,B 0,C 180,E1 -19613.566,E2 -19613.566} C_VEL
LIN {X 0,Y 256.013,Z 647.05,A -85,B 0,C 180,E1 -19615.277,E2 -19615.277} C_VEL
LIN {X 0,Y 253.313,Z 655.434,A -85,B 0,C 180,E1 -19617.159,E2 -19617.159} C_VEL
LIN {X 0,Y 250.501,Z 662.708,A -85,B 0,C 180,E1 -19619.197,E2 -19619.197} C_VEL
LIN {X 0,Y 247.523,Z 669.486,A -85,B 0,C 180,E1 -19621.628,E2 -19621.628} C_VEL
LIN {X 0,Y 244.795,Z 674.758,A -85,B 0,C 180,E1 -19624.117,E2 -19624.117} C_VEL
LIN {X 0,Y 242.43,Z 678.713,A -85,B 0,C 180,E1 -19626.66,E2 -19626.66} C_VEL
LIN {X 0,Y 241.061,Z 680.695,A -85,B 0,C 180,E1 -19628.383,E2 -19628.383} C_VEL
LIN {X 0,Y 239.785,Z 682.138,A -85,B 0,C 180,E1 -19630.129,E2 -19630.129} C_VEL
LIN {X 0,Y 238.07,Z 683.484,A -85,B 0,C 180,E1 -19633.054,E2 -19633.054} C_VEL
LIN {X 0,Y 236.955,Z 683.602,A -85,B 0,C 180,E1 -19635.483,E2 -19635.483} C_VEL
LIN {X 0,Y 236.174,Z 682.903,A -85,B 0,C 180,E1 -19637.782,E2 -19637.782} C_VEL
LIN {X 0,Y 235.494,Z 680.655,A -85,B 0,C 180,E1 -19640.986,E2 -19640.986} C_VEL
LIN {X 0,Y 235.301,Z 677.394,A -85,B 0,C 180,E1 -19643.78,E2 -19643.78} C_VEL
LIN {X 0,Y 235.466,Z 672.829,A -85,B 0,C 180,E1 -19646.597,E2 -19646.597} C_VEL
LIN {X 0,Y 235.873,Z 666.8,A -85,B 0,C 180,E1 -19649.418,E2 -19649.418} C_VEL
LIN {X 0,Y 236.514,Z 660.24,A -85,B 0,C 180,E1 -19651.833,E2 -19651.833} C_VEL
LIN {X 0,Y 237.363,Z 652.193,A -85,B 0,C 180,E1 -19654.234,E2 -19654.234} C_VEL
LIN {X 0,Y 238.188,Z 644.279,A -85,B 0,C 180,E1 -19656.166,E2 -19656.166} C_VEL
LIN {X 0,Y 239.311,Z 633.217,A -85,B 0,C 180,E1 -19658.346,E2 -19658.346} C_VEL
LIN {X 0,Y 240.297,Z 622.396,A -85,B 0,C 180,E1 -19660.049,E2 -19660.049} C_VEL
LIN {X 0,Y 241.22,Z 609.484,A -85,B 0,C 180,E1 -19661.625,E2 -19661.625} C_VEL
LIN {X 0,Y 241.924,Z 597.11,A -85,B 0,C 180,E1 -19662.753,E2 -19662.753} C_VEL
LIN {X 0,Y 242.376,Z 583.14,A -85,B 0,C 180,E1 -19663.642,E2 -19663.642} C_VEL
LIN {X 0,Y 242.44,Z 570.226,A -85,B 0,C 180,E1 -19664.19,E2 -19664.19} C_VEL
LIN {X 0,Y 235.168,Z 547.013,A -85,B 0,C 180,E1 -19665.574,E2 -19665.574} C_VEL
LIN {X 0,Y 235.011,Z 546.145,A -85,B 0,C 180,E1 -19665.868,E2 -19665.868} C_VEL
LIN {X 0,Y 234.945,Z 546.032,A -85,B 0,C 180,E1 -19668.847,E2 -19668.847} C_VEL
LIN {X 0,Y 234.947,Z 546.033,A -85,B 0,C 180,E1 -19673.256,E2 -19673.256} C_VEL
LIN {X 0,Y 234.962,Z 546.031,A -85,B 0,C 180,E1 -19677.426,E2 -19677.426} C_VEL
LIN {X 0,Y 234.954,Z 546.032,A -85,B 0,C 180,E1 -19681.407,E2 -19681.407} C_VEL
LIN {X 0,Y 234.99,Z 546.026,A -85,B 0,C 180,E1 -19685.248,E2 -19685.248} C_VEL
LIN {X 0,Y 235.01,Z 546.022,A -85,B 0,C 180,E1 -19688.97,E2 -19688.97} C_VEL
LIN {X 0,Y 235.059,Z 546.014,A -85,B 0,C 180,E1 -19693.093,E2 -19693.093} C_VEL
LIN {X 0,Y 235.114,Z 546.011,A -85,B 0,C 180,E1 -19697.922,E2 -19697.922} C_VEL
LIN {X 0,Y 235.326,Z 545.983,A -85,B 0,C 180,E1 -19701.413,E2 -19701.413} C_VEL
LIN {X 0,Y 235.363,Z 545.975,A -85,B 0,C 180,E1 -19703.14,E2 -19703.14} C_VEL
LIN {X 0,Y 235.599,Z 545.948,A -85,B 0,C 180,E1 -19708.291,E2 -19708.291} C_VEL
LIN {X 0,Y 235.599,Z 545.949,A -85,B 0,C 180,E1 -19711.709,E2 -19711.709} C_VEL
LIN {X 0,Y 235.364,Z 545.977,A -85,B 0,C 180,E1 -19716.86,E2 -19716.86} C_VEL
LIN {X 0,Y 235.218,Z 545.994,A -85,B 0,C 180,E1 -19720.327,E2 -19720.327} C_VEL
LIN {X 0,Y 235.118,Z 546.01,A -85,B 0,C 180,E1 -19725.606,E2 -19725.606} C_VEL
LIN {X 0,Y 235.012,Z 546.018,A -85,B 0,C 180,E1 -19729.205,E2 -19729.205} C_VEL
LIN {X 0,Y 234.956,Z 546.028,A -85,B 0,C 180,E1 -19732.883,E2 -19732.883} C_VEL
LIN {X 0,Y 234.97,Z 546.025,A -85,B 0,C 180,E1 -19736.657,E2 -19736.657} C_VEL
LIN {X 0,Y 234.925,Z 546.032,A -85,B 0,C 180,E1 -19740.568,E2 -19740.568} C_VEL
LIN {X 0,Y 234.962,Z 546.027,A -85,B 0,C 180,E1 -19744.632,E2 -19744.632} C_VEL
LIN {X 0,Y 234.968,Z 546.026,A -85,B 0,C 180,E1 -19748.951,E2 -19748.951} C_VEL
LIN {X 0,Y 234.965,Z 546.027,A -85,B 0,C 180,E1 -19753.467,E2 -19753.467} C_VEL
LIN {X 0,Y 234.913,Z 546.036,A -85,B 0,C 180,E1 -19758.411,E2 -19758.411} C_VEL
LIN {X 0,Y 234.919,Z 546.033,A -85,B 0,C 180,E1 -19761.078,E2 -19761.078} C_VEL
LIN {X 0,Y 234.959,Z 546.025,A -85,B 0,C 180,E1 -19765.366,E2 -19765.366} C_VEL
LIN {X 0,Y 234.967,Z 546.031,A -85,B 0,C 180,E1 -19770.157,E2 -19770.157} C_VEL
LIN {X 0,Y 234.992,Z 546.022,A -85,B 0,C 180,E1 -19773.793,E2 -19773.793} C_VEL
LIN {X 0,Y 235.025,Z 546.02,A -85,B 0,C 180,E1 -19778.97,E2 -19778.97} C_VEL
LIN {X 0,Y 235.094,Z 546.009,A -85,B 0,C 180,E1 -19783.058,E2 -19783.058} C_VEL
LIN {X 0,Y 235.114,Z 546.01,A -85,B 0,C 180,E1 -19787.921,E2 -19787.921} C_VEL
LIN {X 0,Y 235.373,Z 545.973,A -85,B 0,C 180,E1 -19791.413,E2 -19791.413} C_VEL
LIN {X 0,Y 235.4,Z 545.972,A -85,B 0,C 180,E1 -19793.141,E2 -19793.141} C_VEL
LIN {X 0,Y 235.591,Z 545.952,A -85,B 0,C 180,E1 -19798.29,E2 -19798.29} C_VEL
LIN {X 0,Y 235.591,Z 545.947,A -85,B 0,C 180,E1 -19801.709,E2 -19801.709} C_VEL
LIN {X 0,Y 235.397,Z 545.974,A -85,B 0,C 180,E1 -19806.858,E2 -19806.858} C_VEL
LIN {X 0,Y 235.233,Z 545.993,A -85,B 0,C 180,E1 -19810.326,E2 -19810.326} C_VEL
LIN {X 0,Y 235.107,Z 546.009,A -85,B 0,C 180,E1 -19815.606,E2 -19815.606} C_VEL
LIN {X 0,Y 235.002,Z 546.022,A -85,B 0,C 180,E1 -19819.206,E2 -19819.206} C_VEL
LIN {X 0,Y 234.948,Z 546.032,A -85,B 0,C 180,E1 -19822.884,E2 -19822.884} C_VEL
LIN {X 0,Y 234.965,Z 546.028,A -85,B 0,C 180,E1 -19826.657,E2 -19826.657} C_VEL
LIN {X 0,Y 234.927,Z 546.034,A -85,B 0,C 180,E1 -19830.568,E2 -19830.568} C_VEL
LIN {X 0,Y 234.922,Z 546.035,A -85,B 0,C 180,E1 -19834.639,E2 -19834.639} C_VEL
LIN {X 0,Y 234.938,Z 546.034,A -85,B 0,C 180,E1 -19838.945,E2 -19838.945} C_VEL
LIN {X 0,Y 234.886,Z 546.037,A -85,B 0,C 180,E1 -19843.486,E2 -19843.486} C_VEL
LIN {X 0,Y 234.886,Z 546.039,A -85,B 0,C 180,E1 -19846.515,E2 -19846.515} C_VEL
LIN {X 0,Y 234.879,Z 546.038,A -85,B 0,C 180,E1 -19849.383,E2 -19849.383} C_VEL
LIN {X 0,Y 234.218,Z 546.132,A -85,B 0,C 180,E1 -19850.363,E2 -19850.363} C_VEL
LIN {X 0,Y 231.495,Z 546.46,A -85,B 0,C 180,E1 -19851.916,E2 -19851.916} C_VEL
LIN {X 0,Y 229.339,Z 547.43,A -85,B 0,C 180,E1 -19853.134,E2 -19853.134} C_VEL
LIN {X 0,Y 228.539,Z 548.954,A -85,B 0,C 180,E1 -19854.124,E2 -19854.124} C_VEL
LIN {X 0,Y 228.571,Z 549.424,A -85,B 0,C 180,E1 -19854.344,E2 -19854.344} C_VEL
LIN {X 0,Y 230.934,Z 561.147,A -85,B 0,C 180,E1 -19859.353,E2 -19859.353} C_VEL
LIN {X 0,Y 230.597,Z 564.711,A -85,B 0,C 180,E1 -19860.815,E2 -19860.815} C_VEL
LIN {X 0,Y 228.774,Z 576.278,A -85,B 0,C 180,E1 -19865.499,E2 -19865.499} C_VEL
LIN {X 0,Y 228.791,Z 580.497,A -85,B 0,C 180,E1 -19865.802,E2 -19865.802} C_VEL
LIN {X 0,Y 230.908,Z 624.411,A -85,B 0,C 180,E1 -19868.039,E2 -19868.039} C_VEL
LIN {X 0,Y 232.754,Z 655.857,A -85,B 0,C 180,E1 -19869.645,E2 -19869.645} C_VEL
LIN {X 0,Y 232.17,Z 668.774,A -85,B 0,C 180,E1 -19870.411,E2 -19870.411} C_VEL
LIN {X 0,Y 231.465,Z 680.196,A -85,B 0,C 180,E1 -19871.409,E2 -19871.409} C_VEL
LIN {X 0,Y 230.472,Z 691.181,A -85,B 0,C 180,E1 -19872.704,E2 -19872.704} C_VEL
LIN {X 0,Y 229.239,Z 702.385,A -85,B 0,C 180,E1 -19874.44,E2 -19874.44} C_VEL
LIN {X 0,Y 228.45,Z 711.373,A -85,B 0,C 180,E1 -19876.207,E2 -19876.207} C_VEL
LIN {X 0,Y 227.683,Z 720.298,A -85,B 0,C 180,E1 -19878.426,E2 -19878.426} C_VEL
LIN {X 0,Y 227.35,Z 727.426,A -85,B 0,C 180,E1 -19880.66,E2 -19880.66} C_VEL
LIN {X 0,Y 227.382,Z 733.117,A -85,B 0,C 180,E1 -19882.898,E2 -19882.898} C_VEL
LIN {X 0,Y 227.745,Z 738.374,A -85,B 0,C 180,E1 -19885.575,E2 -19885.575} C_VEL
LIN {X 0,Y 228.191,Z 742.016,A -85,B 0,C 180,E1 -19888.235,E2 -19888.235} C_VEL
LIN {X 0,Y 228.496,Z 743.685,A -85,B 0,C 180,E1 -19890,E2 -19890} C_VEL
LIN {X 0,Y 227.866,Z 744.554,A -85,B 0,C 180,E1 -19891.767,E2 -19891.767} C_VEL
LIN {X 0,Y 227.268,Z 744.93,A -85,B 0,C 180,E1 -19893.546,E2 -19893.546} C_VEL
LIN {X 0,Y 226.892,Z 744.779,A -85,B 0,C 180,E1 -19895.332,E2 -19895.332} C_VEL
LIN {X 0,Y 226.576,Z 744.143,A -85,B 0,C 180,E1 -19897.127,E2 -19897.127} C_VEL
LIN {X 0,Y 226.496,Z 743.025,A -85,B 0,C 180,E1 -19898.925,E2 -19898.925} C_VEL
LIN {X 0,Y 226.896,Z 740.458,A -85,B 0,C 180,E1 -19901.615,E2 -19901.615} C_VEL
LIN {X 0,Y 227.912,Z 736.766,A -85,B 0,C 180,E1 -19904.281,E2 -19904.281} C_VEL
LIN {X 0,Y 229.826,Z 731.932,A -85,B 0,C 180,E1 -19906.888,E2 -19906.888} C_VEL
LIN {X 0,Y 232.231,Z 725.704,A -85,B 0,C 180,E1 -19909.444,E2 -19909.444} C_VEL
LIN {X 0,Y 235.387,Z 717.892,A -85,B 0,C 180,E1 -19911.913,E2 -19911.913} C_VEL
LIN {X 0,Y 239.25,Z 708.089,A -85,B 0,C 180,E1 -19914.283,E2 -19914.283} C_VEL
LIN {X 0,Y 242.84,Z 697.941,A -85,B 0,C 180,E1 -19916.189,E2 -19916.189} C_VEL
LIN {X 0,Y 246.479,Z 686.558,A -85,B 0,C 180,E1 -19917.833,E2 -19917.833} C_VEL
LIN {X 0,Y 249.855,Z 674.481,A -85,B 0,C 180,E1 -19919.142,E2 -19919.142} C_VEL
LIN {X 0,Y 252.948,Z 659.981,A -85,B 0,C 180,E1 -19920.316,E2 -19920.316} C_VEL
LIN {X 0,Y 254.315,Z 645.583,A -85,B 0,C 180,E1 -19921.321,E2 -19921.321} C_VEL
LIN {X 0,Y 254.328,Z 631.338,A -85,B 0,C 180,E1 -19922.257,E2 -19922.257} C_VEL
LIN {X 0,Y 253.402,Z 615.657,A -85,B 0,C 180,E1 -19923.559,E2 -19923.559} C_VEL
LIN {X 0,Y 252.011,Z 601.351,A -85,B 0,C 180,E1 -19925.013,E2 -19925.013} C_VEL
LIN {X 0,Y 250.304,Z 588.506,A -85,B 0,C 180,E1 -19926.55,E2 -19926.55} C_VEL
LIN {X 0,Y 247.55,Z 580.983,A -85,B 0,C 180,E1 -19928.217,E2 -19928.217} C_VEL
LIN {X 0,Y 245.096,Z 574.453,A -85,B 0,C 180,E1 -19929.857,E2 -19929.857} C_VEL
LIN {X 0,Y 242.06,Z 566.965,A -85,B 0,C 180,E1 -19932.129,E2 -19932.129} C_VEL
LIN {X 0,Y 239.415,Z 561.729,A -85,B 0,C 180,E1 -19934.375,E2 -19934.375} C_VEL
LIN {X 0,Y 237.822,Z 558.713,A -85,B 0,C 180,E1 -19935.998,E2 -19935.998} C_VEL
LIN {X 0,Y 235.004,Z 556.502,A -85,B 0,C 180,E1 -19939.142,E2 -19939.142} C_VEL
LIN {X 0,Y 233.545,Z 553.586,A -85,B 0,C 180,E1 -19942.43,E2 -19942.43} C_VEL
LIN {X 0,Y 233.004,Z 553.058,A -85,B 0,C 180,E1 -19945.035,E2 -19945.035} C_VEL
LIN {X 0,Y 233.323,Z 553.394,A -85,B 0,C 180,E1 -19948.442,E2 -19948.442} C_VEL
LIN {X 0,Y 233.902,Z 554.512,A -85,B 0,C 180,E1 -19950.178,E2 -19950.178} C_VEL
LIN {X 0,Y 236.007,Z 557.501,A -85,B 0,C 180,E1 -19953.624,E2 -19953.624} C_VEL
LIN {X 0,Y 238.015,Z 558.862,A -85,B 0,C 180,E1 -19955.641,E2 -19955.641} C_VEL
LIN {X 0,Y 239.726,Z 562.009,A -85,B 0,C 180,E1 -19957.257,E2 -19957.257} C_VEL
LIN {X 0,Y 242.218,Z 564.408,A -85,B 0,C 180,E1 -19959.036,E2 -19959.036} C_VEL
LIN {X 0,Y 244.342,Z 567.708,A -85,B 0,C 180,E1 -19960.471,E2 -19960.471} C_VEL
LIN {X 0,Y 245.872,Z 569.419,A -85,B 0,C 180,E1 -19961.35,E2 -19961.35} C_VEL
LIN {X 0,Y 249.061,Z 574.104,A -85,B 0,C 180,E1 -19963.073,E2 -19963.073} C_VEL
LIN {X 0,Y 253.615,Z 581.051,A -85,B 0,C 180,E1 -19965.209,E2 -19965.209} C_VEL
LIN {X 0,Y 257.721,Z 588.145,A -85,B 0,C 180,E1 -19966.948,E2 -19966.948} C_VEL
LIN {X 0,Y 260.366,Z 593.714,A -85,B 0,C 180,E1 -19968.031,E2 -19968.031} C_VEL
LIN {X 0,Y 259.507,Z 605.862,A -85,B 0,C 180,E1 -19968.806,E2 -19968.806} C_VEL
LIN {X 0,Y 257.978,Z 617.414,A -85,B 0,C 180,E1 -19969.801,E2 -19969.801} C_VEL
LIN {X 0,Y 255.916,Z 628.73,A -85,B 0,C 180,E1 -19971.069,E2 -19971.069} C_VEL
LIN {X 0,Y 253.326,Z 639.434,A -85,B 0,C 180,E1 -19972.629,E2 -19972.629} C_VEL
LIN {X 0,Y 250.488,Z 648.907,A -85,B 0,C 180,E1 -19974.365,E2 -19974.365} C_VEL
LIN {X 0,Y 247.388,Z 657.604,A -85,B 0,C 180,E1 -19976.41,E2 -19976.41} C_VEL
LIN {X 0,Y 244.069,Z 665.579,A -85,B 0,C 180,E1 -19978.763,E2 -19978.763} C_VEL
LIN {X 0,Y 240.763,Z 672.285,A -85,B 0,C 180,E1 -19981.391,E2 -19981.391} C_VEL
LIN {X 0,Y 238.55,Z 676.196,A -85,B 0,C 180,E1 -19983.379,E2 -19983.379} C_VEL
LIN {X 0,Y 236.014,Z 680.059,A -85,B 0,C 180,E1 -19985.983,E2 -19985.983} C_VEL
LIN {X 0,Y 233.832,Z 682.767,A -85,B 0,C 180,E1 -19988.644,E2 -19988.644} C_VEL
LIN {X 0,Y 232.534,Z 683.943,A -85,B 0,C 180,E1 -19990.449,E2 -19990.449} C_VEL
LIN {X 0,Y 230.978,Z 684.776,A -85,B 0,C 180,E1 -19993.184,E2 -19993.184} C_VEL
LIN {X 0,Y 229.736,Z 684.533,A -85,B 0,C 180,E1 -19995.982,E2 -19995.982} C_VEL
LIN {X 0,Y 229.077,Z 683.698,A -85,B 0,C 180,E1 -19998.002,E2 -19998.002} C_VEL
LIN {X 0,Y 228.662,Z 682.479,A -85,B 0,C 180,E1 -19999.761,E2 -19999.761} C_VEL
LIN {X 0,Y 228.281,Z 679.688,A -85,B 0,C 180,E1 -20002.546,E2 -20002.546} C_VEL
LIN {X 0,Y 228.286,Z 675.414,A -85,B 0,C 180,E1 -20005.532,E2 -20005.532} C_VEL
LIN {X 0,Y 228.644,Z 669.742,A -85,B 0,C 180,E1 -20008.454,E2 -20008.454} C_VEL
LIN {X 0,Y 229.174,Z 663.914,A -85,B 0,C 180,E1 -20010.835,E2 -20010.835} C_VEL
LIN {X 0,Y 229.944,Z 656.257,A -85,B 0,C 180,E1 -20013.378,E2 -20013.378} C_VEL
LIN {X 0,Y 230.933,Z 646.873,A -85,B 0,C 180,E1 -20015.863,E2 -20015.863} C_VEL
LIN {X 0,Y 232.01,Z 636.654,A -85,B 0,C 180,E1 -20018.041,E2 -20018.041} C_VEL
LIN {X 0,Y 233.01,Z 625.93,A -85,B 0,C 180,E1 -20019.863,E2 -20019.863} C_VEL
LIN {X 0,Y 233.998,Z 613.736,A -85,B 0,C 180,E1 -20021.502,E2 -20021.502} C_VEL
LIN {X 0,Y 234.802,Z 601.19,A -85,B 0,C 180,E1 -20022.772,E2 -20022.772} C_VEL
LIN {X 0,Y 235.285,Z 588.581,A -85,B 0,C 180,E1 -20023.698,E2 -20023.698} C_VEL
LIN {X 0,Y 235.516,Z 571.612,A -85,B 0,C 180,E1 -20024.491,E2 -20024.491} C_VEL
LIN {X 0,Y 228.11,Z 547.798,A -85,B 0,C 180,E1 -20025.963,E2 -20025.963} C_VEL
LIN {X 0,Y 227.964,Z 546.971,A -85,B 0,C 180,E1 -20026.31,E2 -20026.31} C_VEL
LIN {X 0,Y 227.905,Z 546.908,A -85,B 0,C 180,E1 -20030.439,E2 -20030.439} C_VEL
LIN {X 0,Y 227.902,Z 546.908,A -85,B 0,C 180,E1 -20034.133,E2 -20034.133} C_VEL
LIN {X 0,Y 227.875,Z 546.911,A -85,B 0,C 180,E1 -20038.379,E2 -20038.379} C_VEL
LIN {X 0,Y 227.889,Z 546.908,A -85,B 0,C 180,E1 -20042.446,E2 -20042.446} C_VEL
LIN {X 0,Y 227.917,Z 546.904,A -85,B 0,C 180,E1 -20046.368,E2 -20046.368} C_VEL
LIN {X 0,Y 227.936,Z 546.903,A -85,B 0,C 180,E1 -20050.175,E2 -20050.175} C_VEL
LIN {X 0,Y 228.027,Z 546.891,A -85,B 0,C 180,E1 -20053.896,E2 -20053.896} C_VEL
LIN {X 0,Y 228.071,Z 546.889,A -85,B 0,C 180,E1 -20057.544,E2 -20057.544} C_VEL
LIN {X 0,Y 228.264,Z 546.861,A -85,B 0,C 180,E1 -20061.145,E2 -20061.145} C_VEL
LIN {X 0,Y 228.315,Z 546.852,A -85,B 0,C 180,E1 -20062.928,E2 -20062.928} C_VEL
LIN {X 0,Y 228.557,Z 546.826,A -85,B 0,C 180,E1 -20068.238,E2 -20068.238} C_VEL
LIN {X 0,Y 228.558,Z 546.826,A -85,B 0,C 180,E1 -20071.762,E2 -20071.762} C_VEL
LIN {X 0,Y 228.315,Z 546.856,A -85,B 0,C 180,E1 -20077.073,E2 -20077.073} C_VEL
LIN {X 0,Y 228.15,Z 546.873,A -85,B 0,C 180,E1 -20080.651,E2 -20080.651} C_VEL
LIN {X 0,Y 228.069,Z 546.888,A -85,B 0,C 180,E1 -20084.272,E2 -20084.272} C_VEL
LIN {X 0,Y 228.007,Z 546.894,A -85,B 0,C 180,E1 -20087.953,E2 -20087.953} C_VEL
LIN {X 0,Y 227.92,Z 546.906,A -85,B 0,C 180,E1 -20092.32,E2 -20092.32} C_VEL
LIN {X 0,Y 227.944,Z 546.9,A -85,B 0,C 180,E1 -20096.601,E2 -20096.601} C_VEL
LIN {X 0,Y 227.899,Z 546.909,A -85,B 0,C 180,E1 -20100.29,E2 -20100.29} C_VEL
LIN {X 0,Y 227.892,Z 546.91,A -85,B 0,C 180,E1 -20103.717,E2 -20103.717} C_VEL
LIN {X 0,Y 227.873,Z 546.911,A -85,B 0,C 180,E1 -20108.084,E2 -20108.084} C_VEL
LIN {X 0,Y 227.91,Z 546.906,A -85,B 0,C 180,E1 -20112.718,E2 -20112.718} C_VEL
LIN {X 0,Y 227.843,Z 546.914,A -85,B 0,C 180,E1 -20117.756,E2 -20117.756} C_VEL
LIN {X 0,Y 227.848,Z 546.916,A -85,B 0,C 180,E1 -20121.909,E2 -20121.909} C_VEL
LIN {X 0,Y 227.887,Z 546.911,A -85,B 0,C 180,E1 -20126.28,E2 -20126.28} C_VEL
LIN {X 0,Y 227.917,Z 546.907,A -85,B 0,C 180,E1 -20130.437,E2 -20130.437} C_VEL
LIN {X 0,Y 227.927,Z 546.905,A -85,B 0,C 180,E1 -20134.425,E2 -20134.425} C_VEL
LIN {X 0,Y 227.989,Z 546.9,A -85,B 0,C 180,E1 -20138.289,E2 -20138.289} C_VEL
LIN {X 0,Y 228.033,Z 546.889,A -85,B 0,C 180,E1 -20142.824,E2 -20142.824} C_VEL
LIN {X 0,Y 228.071,Z 546.886,A -85,B 0,C 180,E1 -20147.542,E2 -20147.542} C_VEL
LIN {X 0,Y 228.302,Z 546.854,A -85,B 0,C 180,E1 -20151.145,E2 -20151.145} C_VEL
LIN {X 0,Y 228.351,Z 546.851,A -85,B 0,C 180,E1 -20152.928,E2 -20152.928} C_VEL
LIN {X 0,Y 228.55,Z 546.828,A -85,B 0,C 180,E1 -20158.237,E2 -20158.237} C_VEL
LIN {X 0,Y 228.55,Z 546.824,A -85,B 0,C 180,E1 -20161.762,E2 -20161.762} C_VEL
LIN {X 0,Y 228.349,Z 546.851,A -85,B 0,C 180,E1 -20167.071,E2 -20167.071} C_VEL
LIN {X 0,Y 228.159,Z 546.877,A -85,B 0,C 180,E1 -20170.65,E2 -20170.65} C_VEL
LIN {X 0,Y 228.058,Z 546.889,A -85,B 0,C 180,E1 -20174.272,E2 -20174.272} C_VEL
LIN {X 0,Y 227.998,Z 546.892,A -85,B 0,C 180,E1 -20177.953,E2 -20177.953} C_VEL
LIN {X 0,Y 227.912,Z 546.907,A -85,B 0,C 180,E1 -20182.321,E2 -20182.321} C_VEL
LIN {X 0,Y 227.938,Z 546.903,A -85,B 0,C 180,E1 -20186.603,E2 -20186.603} C_VEL
LIN {X 0,Y 227.904,Z 546.907,A -85,B 0,C 180,E1 -20190.296,E2 -20190.296} C_VEL
LIN {X 0,Y 227.873,Z 546.91,A -85,B 0,C 180,E1 -20193.721,E2 -20193.721} C_VEL
LIN {X 0,Y 227.839,Z 546.914,A -85,B 0,C 180,E1 -20198.091,E2 -20198.091} C_VEL
LIN {X 0,Y 227.809,Z 546.921,A -85,B 0,C 180,E1 -20202.742,E2 -20202.742} C_VEL
LIN {X 0,Y 227.813,Z 546.92,A -85,B 0,C 180,E1 -20207.259,E2 -20207.259} C_VEL
LIN {X 0,Y 227.951,Z 546.901,A -85,B 0,C 180,E1 -20211.931,E2 -20211.931} C_VEL
LIN {X 0,Y 228.133,Z 547.133,A -85,B 0,C 180,E1 -20213.305,E2 -20213.305} C_VEL
LIN {X 0,Y 228.571,Z 549.424,A -85,B 0,C 180,E1 -20214.344,E2 -20214.344} C_VEL
LIN {X 0,Y 228.495,Z 552.425,A -85,B 0,C 180,E1 -20215.624,E2 -20215.624} C_VEL
LIN {X 0,Y 227.565,Z 555.475,A -85,B 0,C 180,E1 -20216.886,E2 -20216.886} C_VEL
LIN {X 0,Y 223.324,Z 565.72,A -85,B 0,C 180,E1 -20221.146,E2 -20221.146} C_VEL
LIN {X 0,Y 221.802,Z 575.07,A -85,B 0,C 180,E1 -20225.051,E2 -20225.051} C_VEL
LIN {X 0,Y 221.881,Z 580.974,A -85,B 0,C 180,E1 -20225.435,E2 -20225.435} C_VEL
LIN {X 0,Y 223.744,Z 621.865,A -85,B 0,C 180,E1 -20227.608,E2 -20227.608} C_VEL
LIN {X 0,Y 225.736,Z 655.779,A -85,B 0,C 180,E1 -20229.398,E2 -20229.398} C_VEL
LIN {X 0,Y 225.087,Z 669.338,A -85,B 0,C 180,E1 -20230.269,E2 -20230.269} C_VEL
LIN {X 0,Y 224.241,Z 682.025,A -85,B 0,C 180,E1 -20231.499,E2 -20231.499} C_VEL
LIN {X 0,Y 223.23,Z 692.267,A -85,B 0,C 180,E1 -20232.833,E2 -20232.833} C_VEL
LIN {X 0,Y 222.046,Z 702.987,A -85,B 0,C 180,E1 -20234.629,E2 -20234.629} C_VEL
LIN {X 0,Y 221.229,Z 712.563,A -85,B 0,C 180,E1 -20236.684,E2 -20236.684} C_VEL
LIN {X 0,Y 220.511,Z 720.992,A -85,B 0,C 180,E1 -20238.976,E2 -20238.976} C_VEL
LIN {X 0,Y 220.305,Z 728.267,A -85,B 0,C 180,E1 -20241.466,E2 -20241.466} C_VEL
LIN {X 0,Y 220.46,Z 733.205,A -85,B 0,C 180,E1 -20243.594,E2 -20243.594} C_VEL
LIN {X 0,Y 220.909,Z 738.102,A -85,B 0,C 180,E1 -20246.352,E2 -20246.352} C_VEL
LIN {X 0,Y 221.193,Z 740.514,A -85,B 0,C 180,E1 -20248.179,E2 -20248.179} C_VEL
LIN {X 0,Y 221.518,Z 742.272,A -85,B 0,C 180,E1 -20250,E2 -20250} C_VEL
LIN {X 0,Y 220.848,Z 743.266,A -85,B 0,C 180,E1 -20251.823,E2 -20251.823} C_VEL
LIN {X 0,Y 220.227,Z 743.698,A -85,B 0,C 180,E1 -20253.659,E2 -20253.659} C_VEL
LIN {X 0,Y 219.831,Z 743.679,A -85,B 0,C 180,E1 -20255.503,E2 -20255.503} C_VEL
LIN {X 0,Y 219.505,Z 743.123,A -85,B 0,C 180,E1 -20257.358,E2 -20257.358} C_VEL
LIN {X 0,Y 219.458,Z 742.128,A -85,B 0,C 180,E1 -20259.214,E2 -20259.214} C_VEL
LIN {X 0,Y 219.686,Z 740.644,A -85,B 0,C 180,E1 -20261.066,E2 -20261.066} C_VEL
LIN {X 0,Y 220.542,Z 737.542,A -85,B 0,C 180,E1 -20263.827,E2 -20263.827} C_VEL
LIN {X 0,Y 222.291,Z 733.325,A -85,B 0,C 180,E1 -20266.531,E2 -20266.531} C_VEL
LIN {X 0,Y 224.605,Z 727.839,A -85,B 0,C 180,E1 -20269.18,E2 -20269.18} C_VEL
LIN {X 0,Y 227.678,Z 720.909,A -85,B 0,C 180,E1 -20271.741,E2 -20271.741} C_VEL
LIN {X 0,Y 231.282,Z 712.644,A -85,B 0,C 180,E1 -20274.113,E2 -20274.113} C_VEL
LIN {X 0,Y 235.373,Z 702.406,A -85,B 0,C 180,E1 -20276.368,E2 -20276.368} C_VEL
LIN {X 0,Y 239.47,Z 691.169,A -85,B 0,C 180,E1 -20278.244,E2 -20278.244} C_VEL
LIN {X 0,Y 242.559,Z 681.595,A -85,B 0,C 180,E1 -20279.508,E2 -20279.508} C_VEL
LIN {X 0,Y 246.035,Z 669.13,A -85,B 0,C 180,E1 -20280.756,E2 -20280.756} C_VEL
LIN {X 0,Y 248.248,Z 658.277,A -85,B 0,C 180,E1 -20281.628,E2 -20281.628} C_VEL
LIN {X 0,Y 249.635,Z 644.049,A -85,B 0,C 180,E1 -20282.65,E2 -20282.65} C_VEL
LIN {X 0,Y 249.613,Z 629.514,A -85,B 0,C 180,E1 -20283.709,E2 -20283.709} C_VEL
LIN {X 0,Y 248.773,Z 613.728,A -85,B 0,C 180,E1 -20285.127,E2 -20285.127} C_VEL
LIN {X 0,Y 247.267,Z 598.277,A -85,B 0,C 180,E1 -20286.864,E2 -20286.864} C_VEL
LIN {X 0,Y 246.449,Z 592.356,A -85,B 0,C 180,E1 -20287.669,E2 -20287.669} C_VEL
LIN {X 0,Y 244.352,Z 586.202,A -85,B 0,C 180,E1 -20289.053,E2 -20289.053} C_VEL
LIN {X 0,Y 242.112,Z 579.758,A -85,B 0,C 180,E1 -20290.731,E2 -20290.731} C_VEL
LIN {X 0,Y 239.597,Z 572.975,A -85,B 0,C 180,E1 -20292.836,E2 -20292.836} C_VEL
LIN {X 0,Y 237.197,Z 567.932,A -85,B 0,C 180,E1 -20295.048,E2 -20295.048} C_VEL
LIN {X 0,Y 235.895,Z 565.377,A -85,B 0,C 180,E1 -20296.497,E2 -20296.497} C_VEL
LIN {X 0,Y 233.275,Z 563.085,A -85,B 0,C 180,E1 -20299.7,E2 -20299.7} C_VEL
LIN {X 0,Y 232.1,Z 560.461,A -85,B 0,C 180,E1 -20302.729,E2 -20302.729} C_VEL
LIN {X 0,Y 231.677,Z 560.029,A -85,B 0,C 180,E1 -20304.988,E2 -20304.988} C_VEL
LIN {X 0,Y 232.012,Z 560.39,A -85,B 0,C 180,E1 -20308.498,E2 -20308.498} C_VEL
LIN {X 0,Y 232.653,Z 561.991,A -85,B 0,C 180,E1 -20310.496,E2 -20310.496} C_VEL
LIN {X 0,Y 234.865,Z 564.657,A -85,B 0,C 180,E1 -20313.855,E2 -20313.855} C_VEL
LIN {X 0,Y 236.18,Z 565.668,A -85,B 0,C 180,E1 -20315.222,E2 -20315.222} C_VEL
LIN {X 0,Y 237.969,Z 568.783,A -85,B 0,C 180,E1 -20316.964,E2 -20316.964} C_VEL
LIN {X 0,Y 239.976,Z 570.839,A -85,B 0,C 180,E1 -20318.502,E2 -20318.502} C_VEL
LIN {X 0,Y 242.219,Z 574.233,A -85,B 0,C 180,E1 -20320.052,E2 -20320.052} C_VEL
LIN {X 0,Y 243.598,Z 576.037,A -85,B 0,C 180,E1 -20320.921,E2 -20320.921} C_VEL
LIN {X 0,Y 246.448,Z 580.298,A -85,B 0,C 180,E1 -20322.519,E2 -20322.519} C_VEL
LIN {X 0,Y 250.625,Z 587.032,A -85,B 0,C 180,E1 -20324.624,E2 -20324.624} C_VEL
LIN {X 0,Y 254.267,Z 593.603,A -85,B 0,C 180,E1 -20326.281,E2 -20326.281} C_VEL
LIN {X 0,Y 255.767,Z 597.058,A -85,B 0,C 180,E1 -20326.964,E2 -20326.964} C_VEL
LIN {X 0,Y 254.747,Z 608.69,A -85,B 0,C 180,E1 -20327.751,E2 -20327.751} C_VEL
LIN {X 0,Y 253.055,Z 620.163,A -85,B 0,C 180,E1 -20328.79,E2 -20328.79} C_VEL
LIN {X 0,Y 250.671,Z 631.604,A -85,B 0,C 180,E1 -20330.145,E2 -20330.145} C_VEL
LIN {X 0,Y 247.712,Z 642.657,A -85,B 0,C 180,E1 -20331.845,E2 -20331.845} C_VEL
LIN {X 0,Y 244.383,Z 652.642,A -85,B 0,C 180,E1 -20333.81,E2 -20333.81} C_VEL
LIN {X 0,Y 241.371,Z 660.412,A -85,B 0,C 180,E1 -20335.757,E2 -20335.757} C_VEL
LIN {X 0,Y 238.451,Z 666.765,A -85,B 0,C 180,E1 -20337.721,E2 -20337.721} C_VEL
LIN {X 0,Y 235.41,Z 672.572,A -85,B 0,C 180,E1 -20340.001,E2 -20340.001} C_VEL
LIN {X 0,Y 232.183,Z 677.906,A -85,B 0,C 180,E1 -20342.736,E2 -20342.736} C_VEL
LIN {X 0,Y 229.635,Z 681.476,A -85,B 0,C 180,E1 -20345.269,E2 -20345.269} C_VEL
LIN {X 0,Y 227.182,Z 684.197,A -85,B 0,C 180,E1 -20348.145,E2 -20348.145} C_VEL
LIN {X 0,Y 225.286,Z 685.586,A -85,B 0,C 180,E1 -20350.789,E2 -20350.789} C_VEL
LIN {X 0,Y 223.866,Z 686.01,A -85,B 0,C 180,E1 -20353.299,E2 -20353.299} C_VEL
LIN {X 0,Y 222.478,Z 685.3,A -85,B 0,C 180,E1 -20356.518,E2 -20356.518} C_VEL
LIN {X 0,Y 221.919,Z 684.231,A -85,B 0,C 180,E1 -20358.464,E2 -20358.464} C_VEL
LIN {X 0,Y 221.346,Z 681.662,A -85,B 0,C 180,E1 -20361.417,E2 -20361.417} C_VEL
LIN {X 0,Y 221.182,Z 677.829,A -85,B 0,C 180,E1 -20364.399,E2 -20364.399} C_VEL
LIN {X 0,Y 221.402,Z 672.87,A -85,B 0,C 180,E1 -20367.279,E2 -20367.279} C_VEL
LIN {X 0,Y 221.821,Z 667.032,A -85,B 0,C 180,E1 -20369.935,E2 -20369.935} C_VEL
LIN {X 0,Y 222.521,Z 660.071,A -85,B 0,C 180,E1 -20372.475,E2 -20372.475} C_VEL
LIN {X 0,Y 223.48,Z 650.93,A -85,B 0,C 180,E1 -20375.152,E2 -20375.152} C_VEL
LIN {X 0,Y 224.511,Z 641.672,A -85,B 0,C 180,E1 -20377.338,E2 -20377.338} C_VEL
LIN {X 0,Y 225.7,Z 629.912,A -85,B 0,C 180,E1 -20379.553,E2 -20379.553} C_VEL
LIN {X 0,Y 226.604,Z 619.067,A -85,B 0,C 180,E1 -20381.167,E2 -20381.167} C_VEL
LIN {X 0,Y 227.565,Z 605.924,A -85,B 0,C 180,E1 -20382.676,E2 -20382.676} C_VEL
LIN {X 0,Y 228.224,Z 592.385,A -85,B 0,C 180,E1 -20383.788,E2 -20383.788} C_VEL
LIN {X 0,Y 228.477,Z 578.984,A -85,B 0,C 180,E1 -20384.521,E2 -20384.521} C_VEL
LIN {X 0,Y 228.439,Z 572.634,A -85,B 0,C 180,E1 -20384.805,E2 -20384.805} C_VEL
LIN {X 0,Y 221.085,Z 548.649,A -85,B 0,C 180,E1 -20386.335,E2 -20386.335} C_VEL
LIN {X 0,Y 220.927,Z 547.831,A -85,B 0,C 180,E1 -20386.727,E2 -20386.727} C_VEL
LIN {X 0,Y 220.857,Z 547.786,A -85,B 0,C 180,E1 -20390.475,E2 -20390.475} C_VEL
LIN {X 0,Y 220.817,Z 547.792,A -85,B 0,C 180,E1 -20395.049,E2 -20395.049} C_VEL
LIN {X 0,Y 220.87,Z 547.786,A -85,B 0,C 180,E1 -20399.396,E2 -20399.396} C_VEL
LIN {X 0,Y 220.898,Z 547.783,A -85,B 0,C 180,E1 -20403.551,E2 -20403.551} C_VEL
LIN {X 0,Y 220.881,Z 547.784,A -85,B 0,C 180,E1 -20407.554,E2 -20407.554} C_VEL
LIN {X 0,Y 220.962,Z 547.769,A -85,B 0,C 180,E1 -20412.593,E2 -20412.593} C_VEL
LIN {X 0,Y 221.008,Z 547.766,A -85,B 0,C 180,E1 -20417.139,E2 -20417.139} C_VEL
LIN {X 0,Y 221.202,Z 547.74,A -85,B 0,C 180,E1 -20420.86,E2 -20420.86} C_VEL
LIN {X 0,Y 221.134,Z 547.749,A -85,B 0,C 180,E1 -20424.529,E2 -20424.529} C_VEL
LIN {X 0,Y 221.515,Z 547.703,A -85,B 0,C 180,E1 -20428.182,E2 -20428.182} C_VEL
LIN {X 0,Y 221.515,Z 547.703,A -85,B 0,C 180,E1 -20431.818,E2 -20431.818} C_VEL
LIN {X 0,Y 221.252,Z 547.736,A -85,B 0,C 180,E1 -20437.3,E2 -20437.3} C_VEL
LIN {X 0,Y 221.071,Z 547.755,A -85,B 0,C 180,E1 -20440.996,E2 -20440.996} C_VEL
LIN {X 0,Y 221,Z 547.767,A -85,B 0,C 180,E1 -20444.738,E2 -20444.738} C_VEL
LIN {X 0,Y 220.924,Z 547.773,A -85,B 0,C 180,E1 -20448.549,E2 -20448.549} C_VEL
LIN {X 0,Y 220.888,Z 547.781,A -85,B 0,C 180,E1 -20452.675,E2 -20452.675} C_VEL
LIN {X 0,Y 220.886,Z 547.779,A -85,B 0,C 180,E1 -20457.013,E2 -20457.013} C_VEL
LIN {X 0,Y 220.841,Z 547.786,A -85,B 0,C 180,E1 -20460.767,E2 -20460.767} C_VEL
LIN {X 0,Y 220.818,Z 547.788,A -85,B 0,C 180,E1 -20464.951,E2 -20464.951} C_VEL
LIN {X 0,Y 220.857,Z 547.784,A -85,B 0,C 180,E1 -20469.525,E2 -20469.525} C_VEL
LIN {X 0,Y 220.868,Z 547.783,A -85,B 0,C 180,E1 -20472.956,E2 -20472.956} C_VEL
LIN {X 0,Y 220.794,Z 547.794,A -85,B 0,C 180,E1 -20478.052,E2 -20478.052} C_VEL
LIN {X 0,Y 220.824,Z 547.788,A -85,B 0,C 180,E1 -20482.792,E2 -20482.792} C_VEL
LIN {X 0,Y 220.822,Z 547.788,A -85,B 0,C 180,E1 -20487.244,E2 -20487.244} C_VEL
LIN {X 0,Y 220.834,Z 547.787,A -85,B 0,C 180,E1 -20491.485,E2 -20491.485} C_VEL
LIN {X 0,Y 220.871,Z 547.781,A -85,B 0,C 180,E1 -20495.565,E2 -20495.565} C_VEL
LIN {X 0,Y 220.907,Z 547.778,A -85,B 0,C 180,E1 -20499.515,E2 -20499.515} C_VEL
LIN {X 0,Y 221.014,Z 547.762,A -85,B 0,C 180,E1 -20503.369,E2 -20503.369} C_VEL
LIN {X 0,Y 221.103,Z 547.753,A -85,B 0,C 180,E1 -20509.005,E2 -20509.005} C_VEL
LIN {X 0,Y 221.302,Z 547.73,A -85,B 0,C 180,E1 -20512.701,E2 -20512.701} C_VEL
LIN {X 0,Y 221.508,Z 547.705,A -85,B 0,C 180,E1 -20518.181,E2 -20518.181} C_VEL
LIN {X 0,Y 221.508,Z 547.702,A -85,B 0,C 180,E1 -20521.818,E2 -20521.818} C_VEL
LIN {X 0,Y 221.284,Z 547.73,A -85,B 0,C 180,E1 -20527.298,E2 -20527.298} C_VEL
LIN {X 0,Y 221.108,Z 547.754,A -85,B 0,C 180,E1 -20530.994,E2 -20530.994} C_VEL
LIN {X 0,Y 221.011,Z 547.766,A -85,B 0,C 180,E1 -20536.63,E2 -20536.63} C_VEL
LIN {X 0,Y 220.88,Z 547.783,A -85,B 0,C 180,E1 -20540.487,E2 -20540.487} C_VEL
LIN {X 0,Y 220.858,Z 547.787,A -85,B 0,C 180,E1 -20544.435,E2 -20544.435} C_VEL
LIN {X 0,Y 220.832,Z 547.787,A -85,B 0,C 180,E1 -20548.513,E2 -20548.513} C_VEL
LIN {X 0,Y 220.813,Z 547.793,A -85,B 0,C 180,E1 -20552.756,E2 -20552.756} C_VEL
LIN {X 0,Y 220.805,Z 547.791,A -85,B 0,C 180,E1 -20557.278,E2 -20557.278} C_VEL
LIN {X 0,Y 220.767,Z 547.795,A -85,B 0,C 180,E1 -20561.952,E2 -20561.952} C_VEL
LIN {X 0,Y 220.773,Z 547.795,A -85,B 0,C 180,E1 -20565.547,E2 -20565.547} C_VEL
LIN {X 0,Y 220.847,Z 547.787,A -85,B 0,C 180,E1 -20570.473,E2 -20570.473} C_VEL
LIN {X 0,Y 221.052,Z 547.935,A -85,B 0,C 180,E1 -20573.266,E2 -20573.266} C_VEL
LIN {X 0,Y 223.256,Z 558.866,A -85,B 0,C 180,E1 -20578.205,E2 -20578.205} C_VEL
LIN {X 0,Y 223.863,Z 562.659,A -85,B 0,C 180,E1 -20579.848,E2 -20579.848} C_VEL
LIN {X 0,Y 223.324,Z 565.72,A -85,B 0,C 180,E1 -20581.146,E2 -20581.146} C_VEL
LIN {X 0,Y 222.261,Z 567.908,A -85,B 0,C 180,E1 -20582.065,E2 -20582.065} C_VEL
LIN {X 0,Y 218.499,Z 571.529,A -85,B 0,C 180,E1 -20583.59,E2 -20583.59} C_VEL
LIN {X 0,Y 215.943,Z 574.873,A -85,B 0,C 180,E1 -20584.464,E2 -20584.464} C_VEL
LIN {X 0,Y 214.948,Z 577.909,A -85,B 0,C 180,E1 -20584.875,E2 -20584.875} C_VEL
LIN {X 0,Y 214.88,Z 578.843,A -85,B 0,C 180,E1 -20584.939,E2 -20584.939} C_VEL
LIN {X 0,Y 216.421,Z 617.549,A -85,B 0,C 180,E1 -20587.066,E2 -20587.066} C_VEL
LIN {X 0,Y 218.729,Z 655.371,A -85,B 0,C 180,E1 -20589.151,E2 -20589.151} C_VEL
LIN {X 0,Y 218.091,Z 667.746,A -85,B 0,C 180,E1 -20589.978,E2 -20589.978} C_VEL
LIN {X 0,Y 217.335,Z 679.565,A -85,B 0,C 180,E1 -20591.133,E2 -20591.133} C_VEL
LIN {X 0,Y 216.343,Z 690.175,A -85,B 0,C 180,E1 -20592.513,E2 -20592.513} C_VEL
LIN {X 0,Y 215.122,Z 701.082,A -85,B 0,C 180,E1 -20594.364,E2 -20594.364} C_VEL
LIN {X 0,Y 214.352,Z 709.856,A -85,B 0,C 180,E1 -20596.249,E2 -20596.249} C_VEL
LIN {X 0,Y 213.601,Z 718.652,A -85,B 0,C 180,E1 -20598.614,E2 -20598.614} C_VEL
LIN {X 0,Y 213.313,Z 726.355,A -85,B 0,C 180,E1 -20601.263,E2 -20601.263} C_VEL
LIN {X 0,Y 213.448,Z 731.288,A -85,B 0,C 180,E1 -20603.382,E2 -20603.382} C_VEL
LIN {X 0,Y 213.904,Z 736.44,A -85,B 0,C 180,E1 -20606.232,E2 -20606.232} C_VEL
LIN {X 0,Y 214.225,Z 738.958,A -85,B 0,C 180,E1 -20608.12,E2 -20608.12} C_VEL
LIN {X 0,Y 214.53,Z 740.822,A -85,B 0,C 180,E1 -20610,E2 -20610} C_VEL
LIN {X 0,Y 213.831,Z 741.904,A -85,B 0,C 180,E1 -20611.883,E2 -20611.883} C_VEL
LIN {X 0,Y 213.188,Z 742.451,A -85,B 0,C 180,E1 -20613.78,E2 -20613.78} C_VEL
LIN {X 0,Y 212.505,Z 742.224,A -85,B 0,C 180,E1 -20617.182,E2 -20617.182} C_VEL
LIN {X 0,Y 212.442,Z 741.193,A -85,B 0,C 180,E1 -20619.521,E2 -20619.521} C_VEL
LIN {X 0,Y 212.679,Z 739.856,A -85,B 0,C 180,E1 -20621.435,E2 -20621.435} C_VEL
LIN {X 0,Y 213.637,Z 736.962,A -85,B 0,C 180,E1 -20624.283,E2 -20624.283} C_VEL
LIN {X 0,Y 215.493,Z 732.938,A -85,B 0,C 180,E1 -20627.068,E2 -20627.068} C_VEL
LIN {X 0,Y 217.913,Z 727.734,A -85,B 0,C 180,E1 -20629.793,E2 -20629.793} C_VEL
LIN {X 0,Y 221.11,Z 721.165,A -85,B 0,C 180,E1 -20632.421,E2 -20632.421} C_VEL
LIN {X 0,Y 224.838,Z 713.212,A -85,B 0,C 180,E1 -20634.85,E2 -20634.85} C_VEL
LIN {X 0,Y 228.696,Z 704.506,A -85,B 0,C 180,E1 -20636.953,E2 -20636.953} C_VEL
LIN {X 0,Y 232.831,Z 694.218,A -85,B 0,C 180,E1 -20638.878,E2 -20638.878} C_VEL
LIN {X 0,Y 236.468,Z 684.126,A -85,B 0,C 180,E1 -20640.347,E2 -20640.347} C_VEL
LIN {X 0,Y 240.425,Z 671.373,A -85,B 0,C 180,E1 -20641.746,E2 -20641.746} C_VEL
LIN {X 0,Y 243.446,Z 658.435,A -85,B 0,C 180,E1 -20642.853,E2 -20642.853} C_VEL
LIN {X 0,Y 245.054,Z 644.889,A -85,B 0,C 180,E1 -20643.904,E2 -20643.904} C_VEL
LIN {X 0,Y 245.275,Z 632.389,A -85,B 0,C 180,E1 -20644.848,E2 -20644.848} C_VEL
LIN {X 0,Y 244.754,Z 618.129,A -85,B 0,C 180,E1 -20646.14,E2 -20646.14} C_VEL
LIN {X 0,Y 243.533,Z 601.919,A -85,B 0,C 180,E1 -20647.983,E2 -20647.983} C_VEL
LIN {X 0,Y 242.863,Z 596.637,A -85,B 0,C 180,E1 -20648.716,E2 -20648.716} C_VEL
LIN {X 0,Y 241.144,Z 590.961,A -85,B 0,C 180,E1 -20650.054,E2 -20650.054} C_VEL
LIN {X 0,Y 239.19,Z 585.053,A -85,B 0,C 180,E1 -20651.626,E2 -20651.626} C_VEL
LIN {X 0,Y 236.674,Z 577.662,A -85,B 0,C 180,E1 -20654.044,E2 -20654.044} C_VEL
LIN {X 0,Y 235.183,Z 574.317,A -85,B 0,C 180,E1 -20655.614,E2 -20655.614} C_VEL
LIN {X 0,Y 234.034,Z 572.101,A -85,B 0,C 180,E1 -20656.938,E2 -20656.938} C_VEL
LIN {X 0,Y 231.489,Z 569.571,A -85,B 0,C 180,E1 -20660.391,E2 -20660.391} C_VEL
LIN {X 0,Y 230.719,Z 567.411,A -85,B 0,C 180,E1 -20662.837,E2 -20662.837} C_VEL
LIN {X 0,Y 230.314,Z 567.005,A -85,B 0,C 180,E1 -20665.475,E2 -20665.475} C_VEL
LIN {X 0,Y 230.7,Z 567.402,A -85,B 0,C 180,E1 -20668.536,E2 -20668.536} C_VEL
LIN {X 0,Y 232.981,Z 571.293,A -85,B 0,C 180,E1 -20673.254,E2 -20673.254} C_VEL
LIN {X 0,Y 234.384,Z 572.381,A -85,B 0,C 180,E1 -20674.778,E2 -20674.778} C_VEL
LIN {X 0,Y 236.181,Z 575.507,A -85,B 0,C 180,E1 -20676.64,E2 -20676.64} C_VEL
LIN {X 0,Y 237.936,Z 577.531,A -85,B 0,C 180,E1 -20678.068,E2 -20678.068} C_VEL
LIN {X 0,Y 240.561,Z 581.264,A -85,B 0,C 180,E1 -20679.914,E2 -20679.914} C_VEL
LIN {X 0,Y 243.662,Z 586.185,A -85,B 0,C 180,E1 -20681.856,E2 -20681.856} C_VEL
LIN {X 0,Y 247.569,Z 592.817,A -85,B 0,C 180,E1 -20683.978,E2 -20683.978} C_VEL
LIN {X 0,Y 250.979,Z 599.257,A -85,B 0,C 180,E1 -20685.636,E2 -20685.636} C_VEL
LIN {X 0,Y 251.314,Z 600.199,A -85,B 0,C 180,E1 -20685.827,E2 -20685.827} C_VEL
LIN {X 0,Y 250.037,Z 611.982,A -85,B 0,C 180,E1 -20686.692,E2 -20686.692} C_VEL
LIN {X 0,Y 247.976,Z 624.295,A -85,B 0,C 180,E1 -20687.9,E2 -20687.9} C_VEL
LIN {X 0,Y 245.545,Z 634.634,A -85,B 0,C 180,E1 -20689.191,E2 -20689.191} C_VEL
LIN {X 0,Y 242.909,Z 643.757,A -85,B 0,C 180,E1 -20690.631,E2 -20690.631} C_VEL
LIN {X 0,Y 239.69,Z 652.841,A -85,B 0,C 180,E1 -20692.419,E2 -20692.419} C_VEL
LIN {X 0,Y 236.329,Z 660.991,A -85,B 0,C 180,E1 -20694.454,E2 -20694.454} C_VEL
LIN {X 0,Y 233.05,Z 667.784,A -85,B 0,C 180,E1 -20696.543,E2 -20696.543} C_VEL
LIN {X 0,Y 229.457,Z 674.22,A -85,B 0,C 180,E1 -20699.123,E2 -20699.123} C_VEL
LIN {X 0,Y 226.17,Z 679.195,A -85,B 0,C 180,E1 -20701.781,E2 -20701.781} C_VEL
LIN {X 0,Y 223.291,Z 682.893,A -85,B 0,C 180,E1 -20704.514,E2 -20704.514} C_VEL
LIN {X 0,Y 220.09,Z 685.948,A -85,B 0,C 180,E1 -20708.159,E2 -20708.159} C_VEL
LIN {X 0,Y 218.012,Z 687.072,A -85,B 0,C 180,E1 -20711.153,E2 -20711.153} C_VEL
LIN {X 0,Y 216.744,Z 687.122,A -85,B 0,C 180,E1 -20713.41,E2 -20713.41} C_VEL
LIN {X 0,Y 215.986,Z 686.768,A -85,B 0,C 180,E1 -20715.089,E2 -20715.089} C_VEL
LIN {X 0,Y 214.855,Z 685.007,A -85,B 0,C 180,E1 -20718.454,E2 -20718.454} C_VEL
LIN {X 0,Y 214.189,Z 681.449,A -85,B 0,C 180,E1 -20722.17,E2 -20722.17} C_VEL
LIN {X 0,Y 214.133,Z 677.076,A -85,B 0,C 180,E1 -20725.257,E2 -20725.257} C_VEL
LIN {X 0,Y 214.488,Z 670.991,A -85,B 0,C 180,E1 -20728.491,E2 -20728.491} C_VEL
LIN {X 0,Y 215.152,Z 663.635,A -85,B 0,C 180,E1 -20731.511,E2 -20731.511} C_VEL
LIN {X 0,Y 216.01,Z 655.617,A -85,B 0,C 180,E1 -20734.142,E2 -20734.142} C_VEL
LIN {X 0,Y 216.979,Z 646.792,A -85,B 0,C 180,E1 -20736.496,E2 -20736.496} C_VEL
LIN {X 0,Y 218.155,Z 635.507,A -85,B 0,C 180,E1 -20738.895,E2 -20738.895} C_VEL
LIN {X 0,Y 219.232,Z 624.231,A -85,B 0,C 180,E1 -20740.782,E2 -20740.782} C_VEL
LIN {X 0,Y 220.141,Z 612.696,A -85,B 0,C 180,E1 -20742.304,E2 -20742.304} C_VEL
LIN {X 0,Y 220.936,Z 600.253,A -85,B 0,C 180,E1 -20743.543,E2 -20743.543} C_VEL
LIN {X 0,Y 221.416,Z 587.195,A -85,B 0,C 180,E1 -20744.467,E2 -20744.467} C_VEL
LIN {X 0,Y 221.431,Z 573.644,A -85,B 0,C 180,E1 -20745.122,E2 -20745.122} C_VEL
LIN {X 0,Y 214.131,Z 549.933,A -85,B 0,C 180,E1 -20746.674,E2 -20746.674} C_VEL
LIN {X 0,Y 213.912,Z 548.896,A -85,B 0,C 180,E1 -20746.942,E2 -20746.942} C_VEL
LIN {X 0,Y 213.796,Z 548.667,A -85,B 0,C 180,E1 -20749.12,E2 -20749.12} C_VEL
LIN {X 0,Y 213.756,Z 548.672,A -85,B 0,C 180,E1 -20753.715,E2 -20753.715} C_VEL
LIN {X 0,Y 213.798,Z 548.665,A -85,B 0,C 180,E1 -20758.726,E2 -20758.726} C_VEL
LIN {X 0,Y 213.828,Z 548.66,A -85,B 0,C 180,E1 -20762.604,E2 -20762.604} C_VEL
LIN {X 0,Y 213.855,Z 548.656,A -85,B 0,C 180,E1 -20766.954,E2 -20766.954} C_VEL
LIN {X 0,Y 213.92,Z 548.646,A -85,B 0,C 180,E1 -20772.802,E2 -20772.802} C_VEL
LIN {X 0,Y 213.946,Z 548.645,A -85,B 0,C 180,E1 -20776.707,E2 -20776.707} C_VEL
LIN {X 0,Y 214.141,Z 548.62,A -85,B 0,C 180,E1 -20780.556,E2 -20780.556} C_VEL
LIN {X 0,Y 214.095,Z 548.626,A -85,B 0,C 180,E1 -20784.349,E2 -20784.349} C_VEL
LIN {X 0,Y 214.448,Z 548.584,A -85,B 0,C 180,E1 -20788.122,E2 -20788.122} C_VEL
LIN {X 0,Y 214.555,Z 548.569,A -85,B 0,C 180,E1 -20790,E2 -20790} C_VEL
LIN {X 0,Y 214.448,Z 548.583,A -85,B 0,C 180,E1 -20791.878,E2 -20791.878} C_VEL
LIN {X 0,Y 214.193,Z 548.617,A -85,B 0,C 180,E1 -20797.542,E2 -20797.542} C_VEL
LIN {X 0,Y 214.003,Z 548.636,A -85,B 0,C 180,E1 -20801.364,E2 -20801.364} C_VEL
LIN {X 0,Y 213.938,Z 548.647,A -85,B 0,C 180,E1 -20805.236,E2 -20805.236} C_VEL
LIN {X 0,Y 213.84,Z 548.655,A -85,B 0,C 180,E1 -20809.187,E2 -20809.187} C_VEL
LIN {X 0,Y 213.814,Z 548.662,A -85,B 0,C 180,E1 -20813.23,E2 -20813.23} C_VEL
LIN {X 0,Y 213.832,Z 548.658,A -85,B 0,C 180,E1 -20817.449,E2 -20817.449} C_VEL
LIN {X 0,Y 213.772,Z 548.669,A -85,B 0,C 180,E1 -20821.736,E2 -20821.736} C_VEL
LIN {X 0,Y 213.756,Z 548.667,A -85,B 0,C 180,E1 -20826.285,E2 -20826.285} C_VEL
LIN {X 0,Y 213.795,Z 548.664,A -85,B 0,C 180,E1 -20831.105,E2 -20831.105} C_VEL
LIN {X 0,Y 213.809,Z 548.663,A -85,B 0,C 180,E1 -20833.684,E2 -20833.684} C_VEL
LIN {X 0,Y 213.748,Z 548.67,A -85,B 0,C 180,E1 -20836.331,E2 -20836.331} C_VEL
LIN {X 0,Y 213.734,Z 548.672,A -85,B 0,C 180,E1 -20841.335,E2 -20841.335} C_VEL
LIN {X 0,Y 213.767,Z 548.667,A -85,B 0,C 180,E1 -20846.019,E2 -20846.019} C_VEL
LIN {X 0,Y 213.779,Z 548.668,A -85,B 0,C 180,E1 -20850.453,E2 -20850.453} C_VEL
LIN {X 0,Y 213.803,Z 548.663,A -85,B 0,C 180,E1 -20854.701,E2 -20854.701} C_VEL
LIN {X 0,Y 213.838,Z 548.66,A -85,B 0,C 180,E1 -20858.805,E2 -20858.805} C_VEL
LIN {X 0,Y 213.942,Z 548.644,A -85,B 0,C 180,E1 -20862.803,E2 -20862.803} C_VEL
LIN {X 0,Y 213.95,Z 548.647,A -85,B 0,C 180,E1 -20866.706,E2 -20866.706} C_VEL
LIN {X 0,Y 214.164,Z 548.617,A -85,B 0,C 180,E1 -20870.556,E2 -20870.556} C_VEL
LIN {X 0,Y 214.237,Z 548.609,A -85,B 0,C 180,E1 -20872.459,E2 -20872.459} C_VEL
LIN {X 0,Y 214.442,Z 548.585,A -85,B 0,C 180,E1 -20878.121,E2 -20878.121} C_VEL
LIN {X 0,Y 214.546,Z 548.569,A -85,B 0,C 180,E1 -20879.999,E2 -20879.999} C_VEL
LIN {X 0,Y 214.441,Z 548.582,A -85,B 0,C 180,E1 -20881.877,E2 -20881.877} C_VEL
LIN {X 0,Y 214.222,Z 548.609,A -85,B 0,C 180,E1 -20887.54,E2 -20887.54} C_VEL
LIN {X 0,Y 214.04,Z 548.633,A -85,B 0,C 180,E1 -20891.362,E2 -20891.362} C_VEL
LIN {X 0,Y 213.927,Z 548.648,A -85,B 0,C 180,E1 -20895.237,E2 -20895.237} C_VEL
LIN {X 0,Y 213.831,Z 548.659,A -85,B 0,C 180,E1 -20899.187,E2 -20899.187} C_VEL
LIN {X 0,Y 213.807,Z 548.663,A -85,B 0,C 180,E1 -20903.231,E2 -20903.231} C_VEL
LIN {X 0,Y 213.825,Z 548.658,A -85,B 0,C 180,E1 -20907.45,E2 -20907.45} C_VEL
LIN {X 0,Y 213.773,Z 548.667,A -85,B 0,C 180,E1 -20911.736,E2 -20911.736} C_VEL
LIN {X 0,Y 213.74,Z 548.668,A -85,B 0,C 180,E1 -20916.288,E2 -20916.288} C_VEL
LIN {X 0,Y 213.709,Z 548.677,A -85,B 0,C 180,E1 -20921.125,E2 -20921.125} C_VEL
LIN {X 0,Y 213.704,Z 548.675,A -85,B 0,C 180,E1 -20923.678,E2 -20923.678} C_VEL
LIN {X 0,Y 213.706,Z 548.676,A -85,B 0,C 180,E1 -20926.343,E2 -20926.343} C_VEL
LIN {X 0,Y 213.842,Z 548.66,A -85,B 0,C 180,E1 -20931.36,E2 -20931.36} C_VEL
LIN {X 0,Y 214.019,Z 548.825,A -85,B 0,C 180,E1 -20933.328,E2 -20933.328} C_VEL
LIN {X 0,Y 216.391,Z 560.364,A -85,B 0,C 180,E1 -20938.692,E2 -20938.692} C_VEL
LIN {X 0,Y 216.733,Z 562.905,A -85,B 0,C 180,E1 -20939.827,E2 -20939.827} C_VEL
LIN {X 0,Y 214.873,Z 573.841,A -85,B 0,C 180,E1 -20944.578,E2 -20944.578} C_VEL
LIN {X 0,Y 214.882,Z 578.667,A -85,B 0,C 180,E1 -20944.929,E2 -20944.929} C_VEL
LIN {X 0,Y 214.88,Z 578.843,A -85,B 0,C 180,E1 -20944.939,E2 -20944.939} C_VEL
LIN {X 0,Y 214.271,Z 584.636,A -85,B 0,C 180,E1 -20945.212,E2 -20945.212} C_VEL
LIN {X 0,Y 209.425,Z 603.623,A -85,B 0,C 180,E1 -20945.976,E2 -20945.976} C_VEL
LIN {X 0,Y 208.984,Z 609.406,A -85,B 0,C 180,E1 -20946.27,E2 -20946.27} C_VEL
LIN {X 0,Y 211.646,Z 656.324,A -85,B 0,C 180,E1 -20948.97,E2 -20948.97} C_VEL
LIN {X 0,Y 210.991,Z 668.921,A -85,B 0,C 180,E1 -20949.91,E2 -20949.91} C_VEL
LIN {X 0,Y 210.138,Z 681.105,A -85,B 0,C 180,E1 -20951.222,E2 -20951.222} C_VEL
LIN {X 0,Y 208.949,Z 692.546,A -85,B 0,C 180,E1 -20952.884,E2 -20952.884} C_VEL
LIN {X 0,Y 207.749,Z 703.862,A -85,B 0,C 180,E1 -20955.052,E2 -20955.052} C_VEL
LIN {X 0,Y 207.021,Z 712.796,A -85,B 0,C 180,E1 -20957.252,E2 -20957.252} C_VEL
LIN {X 0,Y 206.459,Z 720.753,A -85,B 0,C 180,E1 -20959.705,E2 -20959.705} C_VEL
LIN {X 0,Y 206.393,Z 728.221,A -85,B 0,C 180,E1 -20962.664,E2 -20962.664} C_VEL
LIN {X 0,Y 206.699,Z 733.053,A -85,B 0,C 180,E1 -20965.124,E2 -20965.124} C_VEL
LIN {X 0,Y 207.247,Z 737.315,A -85,B 0,C 180,E1 -20968.057,E2 -20968.057} C_VEL
LIN {X 0,Y 207.558,Z 739.339,A -85,B 0,C 180,E1 -20970,E2 -20970} C_VEL
LIN {X 0,Y 206.846,Z 740.51,A -85,B 0,C 180,E1 -20971.947,E2 -20971.947} C_VEL
LIN {X 0,Y 206.151,Z 741.175,A -85,B 0,C 180,E1 -20973.909,E2 -20973.909} C_VEL
LIN {X 0,Y 205.467,Z 741.16,A -85,B 0,C 180,E1 -20977.282,E2 -20977.282} C_VEL
LIN {X 0,Y 205.418,Z 740.263,A -85,B 0,C 180,E1 -20979.849,E2 -20979.849} C_VEL
LIN {X 0,Y 205.692,Z 739.017,A -85,B 0,C 180,E1 -20981.829,E2 -20981.829} C_VEL
LIN {X 0,Y 206.754,Z 736.319,A -85,B 0,C 180,E1 -20984.77,E2 -20984.77} C_VEL
LIN {X 0,Y 208.696,Z 732.575,A -85,B 0,C 180,E1 -20987.642,E2 -20987.642} C_VEL
LIN {X 0,Y 211.252,Z 727.638,A -85,B 0,C 180,E1 -20990.445,E2 -20990.445} C_VEL
LIN {X 0,Y 215.196,Z 720.168,A -85,B 0,C 180,E1 -20993.582,E2 -20993.582} C_VEL
LIN {X 0,Y 219.356,Z 712.065,A -85,B 0,C 180,E1 -20996.137,E2 -20996.137} C_VEL
LIN {X 0,Y 223.275,Z 703.784,A -85,B 0,C 180,E1 -20998.173,E2 -20998.173} C_VEL
LIN {X 0,Y 227.605,Z 693.644,A -85,B 0,C 180,E1 -21000.116,E2 -21000.116} C_VEL
LIN {X 0,Y 231.949,Z 682.468,A -85,B 0,C 180,E1 -21001.767,E2 -21001.767} C_VEL
LIN {X 0,Y 236.059,Z 669.979,A -85,B 0,C 180,E1 -21003.144,E2 -21003.144} C_VEL
LIN {X 0,Y 238.874,Z 658.379,A -85,B 0,C 180,E1 -21004.171,E2 -21004.171} C_VEL
LIN {X 0,Y 240.669,Z 645.339,A -85,B 0,C 180,E1 -21005.227,E2 -21005.227} C_VEL
LIN {X 0,Y 241.108,Z 633.691,A -85,B 0,C 180,E1 -21006.18,E2 -21006.18} C_VEL
LIN {X 0,Y 240.789,Z 619.957,A -85,B 0,C 180,E1 -21007.474,E2 -21007.474} C_VEL
LIN {X 0,Y 239.895,Z 604.917,A -85,B 0,C 180,E1 -21009.241,E2 -21009.241} C_VEL
LIN {X 0,Y 239.461,Z 600.76,A -85,B 0,C 180,E1 -21009.86,E2 -21009.86} C_VEL
LIN {X 0,Y 237.893,Z 595.326,A -85,B 0,C 180,E1 -21011.183,E2 -21011.183} C_VEL
LIN {X 0,Y 236.457,Z 590.343,A -85,B 0,C 180,E1 -21012.568,E2 -21012.568} C_VEL
LIN {X 0,Y 234.26,Z 583.389,A -85,B 0,C 180,E1 -21014.909,E2 -21014.909} C_VEL
LIN {X 0,Y 232.883,Z 580.146,A -85,B 0,C 180,E1 -21016.544,E2 -21016.544} C_VEL
LIN {X 0,Y 232.089,Z 578.74,A -85,B 0,C 180,E1 -21017.492,E2 -21017.492} C_VEL
LIN {X 0,Y 229.919,Z 576.266,A -85,B 0,C 180,E1 -21020.843,E2 -21020.843} C_VEL
LIN {X 0,Y 229.235,Z 574.227,A -85,B 0,C 180,E1 -21023.296,E2 -21023.296} C_VEL
LIN {X 0,Y 229.134,Z 574.086,A -85,B 0,C 180,E1 -21027.494,E2 -21027.494} C_VEL
LIN {X 0,Y 229.468,Z 574.84,A -85,B 0,C 180,E1 -21029.042,E2 -21029.042} C_VEL
LIN {X 0,Y 231.473,Z 578.189,A -85,B 0,C 180,E1 -21033.065,E2 -21033.065} C_VEL
LIN {X 0,Y 232.59,Z 579.076,A -85,B 0,C 180,E1 -21034.327,E2 -21034.327} C_VEL
LIN {X 0,Y 234.469,Z 582.364,A -85,B 0,C 180,E1 -21036.38,E2 -21036.38} C_VEL
LIN {X 0,Y 235.889,Z 584.096,A -85,B 0,C 180,E1 -21037.58,E2 -21037.58} C_VEL
LIN {X 0,Y 238.933,Z 588.75,A -85,B 0,C 180,E1 -21039.842,E2 -21039.842} C_VEL
LIN {X 0,Y 241.45,Z 593.014,A -85,B 0,C 180,E1 -21041.5,E2 -21041.5} C_VEL
LIN {X 0,Y 244.914,Z 599.232,A -85,B 0,C 180,E1 -21043.476,E2 -21043.476} C_VEL
LIN {X 0,Y 246.97,Z 603.436,A -85,B 0,C 180,E1 -21044.64,E2 -21044.64} C_VEL
LIN {X 0,Y 245.566,Z 615.299,A -85,B 0,C 180,E1 -21045.578,E2 -21045.578} C_VEL
LIN {X 0,Y 243.178,Z 627.541,A -85,B 0,C 180,E1 -21046.845,E2 -21046.845} C_VEL
LIN {X 0,Y 240.508,Z 637.726,A -85,B 0,C 180,E1 -21048.197,E2 -21048.197} C_VEL
LIN {X 0,Y 236.807,Z 648.97,A -85,B 0,C 180,E1 -21050.125,E2 -21050.125} C_VEL
LIN {X 0,Y 233.73,Z 656.716,A -85,B 0,C 180,E1 -21051.789,E2 -21051.789} C_VEL
LIN {X 0,Y 230.218,Z 664.366,A -85,B 0,C 180,E1 -21053.867,E2 -21053.867} C_VEL
LIN {X 0,Y 226.77,Z 670.696,A -85,B 0,C 180,E1 -21056.002,E2 -21056.002} C_VEL
LIN {X 0,Y 223.584,Z 675.859,A -85,B 0,C 180,E1 -21058.199,E2 -21058.199} C_VEL
LIN {X 0,Y 220.091,Z 680.763,A -85,B 0,C 180,E1 -21060.915,E2 -21060.915} C_VEL
LIN {X 0,Y 217.01,Z 684.357,A -85,B 0,C 180,E1 -21063.714,E2 -21063.714} C_VEL
LIN {X 0,Y 215.161,Z 686.07,A -85,B 0,C 180,E1 -21065.624,E2 -21065.624} C_VEL
LIN {X 0,Y 213.005,Z 687.598,A -85,B 0,C 180,E1 -21068.187,E2 -21068.187} C_VEL
LIN {X 0,Y 210.716,Z 688.363,A -85,B 0,C 180,E1 -21071.545,E2 -21071.545} C_VEL
LIN {X 0,Y 209.606,Z 688.158,A -85,B 0,C 180,E1 -21073.575,E2 -21073.575} C_VEL
LIN {X 0,Y 208.711,Z 687.456,A -85,B 0,C 180,E1 -21075.629,E2 -21075.629} C_VEL
LIN {X 0,Y 207.73,Z 685.538,A -85,B 0,C 180,E1 -21078.688,E2 -21078.688} C_VEL
LIN {X 0,Y 207.138,Z 682.343,A -85,B 0,C 180,E1 -21081.915,E2 -21081.915} C_VEL
LIN {X 0,Y 207.055,Z 677.874,A -85,B 0,C 180,E1 -21085.106,E2 -21085.106} C_VEL
LIN {X 0,Y 207.381,Z 671.942,A -85,B 0,C 180,E1 -21088.324,E2 -21088.324} C_VEL
LIN {X 0,Y 207.913,Z 665.628,A -85,B 0,C 180,E1 -21091.031,E2 -21091.031} C_VEL
LIN {X 0,Y 208.729,Z 657.774,A -85,B 0,C 180,E1 -21093.75,E2 -21093.75} C_VEL
LIN {X 0,Y 209.769,Z 648.529,A -85,B 0,C 180,E1 -21096.349,E2 -21096.349} C_VEL
LIN {X 0,Y 210.881,Z 638.182,A -85,B 0,C 180,E1 -21098.674,E2 -21098.674} C_VEL
LIN {X 0,Y 212.022,Z 627.008,A -85,B 0,C 180,E1 -21100.689,E2 -21100.689} C_VEL
LIN {X 0,Y 213.028,Z 614.824,A -85,B 0,C 180,E1 -21102.397,E2 -21102.397} C_VEL
LIN {X 0,Y 213.875,Z 602.577,A -85,B 0,C 180,E1 -21103.705,E2 -21103.705} C_VEL
LIN {X 0,Y 214.433,Z 588.192,A -85,B 0,C 180,E1 -21104.778,E2 -21104.778} C_VEL
LIN {X 0,Y 214.535,Z 575.045,A -85,B 0,C 180,E1 -21105.433,E2 -21105.433} C_VEL
LIN {X 0,Y 207.043,Z 550.578,A -85,B 0,C 180,E1 -21107.082,E2 -21107.082} C_VEL
LIN {X 0,Y 206.822,Z 549.63,A -85,B 0,C 180,E1 -21107.451,E2 -21107.451} C_VEL
LIN {X 0,Y 206.726,Z 549.546,A -85,B 0,C 180,E1 -21112.271,E2 -21112.271} C_VEL
LIN {X 0,Y 206.711,Z 549.549,A -85,B 0,C 180,E1 -21117.046,E2 -21117.046} C_VEL
LIN {X 0,Y 206.769,Z 549.54,A -85,B 0,C 180,E1 -21122.098,E2 -21122.098} C_VEL
LIN {X 0,Y 206.788,Z 549.536,A -85,B 0,C 180,E1 -21126.585,E2 -21126.585} C_VEL
LIN {X 0,Y 206.871,Z 549.525,A -85,B 0,C 180,E1 -21132.197,E2 -21132.197} C_VEL
LIN {X 0,Y 206.886,Z 549.525,A -85,B 0,C 180,E1 -21136.244,E2 -21136.244} C_VEL
LIN {X 0,Y 207.103,Z 549.497,A -85,B 0,C 180,E1 -21140.232,E2 -21140.232} C_VEL
LIN {X 0,Y 207.057,Z 549.504,A -85,B 0,C 180,E1 -21144.156,E2 -21144.156} C_VEL
LIN {X 0,Y 207.384,Z 549.464,A -85,B 0,C 180,E1 -21148.058,E2 -21148.058} C_VEL
LIN {X 0,Y 207.52,Z 549.445,A -85,B 0,C 180,E1 -21150,E2 -21150} C_VEL
LIN {X 0,Y 207.385,Z 549.463,A -85,B 0,C 180,E1 -21151.942,E2 -21151.942} C_VEL
LIN {X 0,Y 207.136,Z 549.496,A -85,B 0,C 180,E1 -21157.8,E2 -21157.8} C_VEL
LIN {X 0,Y 206.929,Z 549.519,A -85,B 0,C 180,E1 -21161.758,E2 -21161.758} C_VEL
LIN {X 0,Y 206.872,Z 549.53,A -85,B 0,C 180,E1 -21165.77,E2 -21165.77} C_VEL
LIN {X 0,Y 206.782,Z 549.537,A -85,B 0,C 180,E1 -21169.869,E2 -21169.869} C_VEL
LIN {X 0,Y 206.75,Z 549.544,A -85,B 0,C 180,E1 -21174.073,E2 -21174.073} C_VEL
LIN {X 0,Y 206.739,Z 549.542,A -85,B 0,C 180,E1 -21178.419,E2 -21178.419} C_VEL
LIN {X 0,Y 206.708,Z 549.547,A -85,B 0,C 180,E1 -21182.955,E2 -21182.955} C_VEL
LIN {X 0,Y 206.727,Z 549.542,A -85,B 0,C 180,E1 -21187.729,E2 -21187.729} C_VEL
LIN {X 0,Y 206.725,Z 549.546,A -85,B 0,C 180,E1 -21191.587,E2 -21191.587} C_VEL
LIN {X 0,Y 206.675,Z 549.549,A -85,B 0,C 180,E1 -21195.569,E2 -21195.569} C_VEL
LIN {X 0,Y 206.669,Z 549.553,A -85,B 0,C 180,E1 -21199.75,E2 -21199.75} C_VEL
LIN {X 0,Y 206.731,Z 549.542,A -85,B 0,C 180,E1 -21204.694,E2 -21204.694} C_VEL
LIN {X 0,Y 206.722,Z 549.545,A -85,B 0,C 180,E1 -21209.338,E2 -21209.338} C_VEL
LIN {X 0,Y 206.733,Z 549.541,A -85,B 0,C 180,E1 -21213.771,E2 -21213.771} C_VEL
LIN {X 0,Y 206.776,Z 549.541,A -85,B 0,C 180,E1 -21218.044,E2 -21218.044} C_VEL
LIN {X 0,Y 206.876,Z 549.526,A -85,B 0,C 180,E1 -21222.196,E2 -21222.196} C_VEL
LIN {X 0,Y 206.892,Z 549.527,A -85,B 0,C 180,E1 -21226.243,E2 -21226.243} C_VEL
LIN {X 0,Y 207.102,Z 549.499,A -85,B 0,C 180,E1 -21230.23,E2 -21230.23} C_VEL
LIN {X 0,Y 207.175,Z 549.487,A -85,B 0,C 180,E1 -21232.201,E2 -21232.201} C_VEL
LIN {X 0,Y 207.379,Z 549.464,A -85,B 0,C 180,E1 -21238.057,E2 -21238.057} C_VEL
LIN {X 0,Y 207.511,Z 549.445,A -85,B 0,C 180,E1 -21239.999,E2 -21239.999} C_VEL
LIN {X 0,Y 207.378,Z 549.462,A -85,B 0,C 180,E1 -21241.941,E2 -21241.941} C_VEL
LIN {X 0,Y 207.163,Z 549.489,A -85,B 0,C 180,E1 -21247.798,E2 -21247.798} C_VEL
LIN {X 0,Y 206.977,Z 549.513,A -85,B 0,C 180,E1 -21251.755,E2 -21251.755} C_VEL
LIN {X 0,Y 206.861,Z 549.527,A -85,B 0,C 180,E1 -21255.77,E2 -21255.77} C_VEL
LIN {X 0,Y 206.758,Z 549.539,A -85,B 0,C 180,E1 -21259.871,E2 -21259.871} C_VEL
LIN {X 0,Y 206.743,Z 549.543,A -85,B 0,C 180,E1 -21264.074,E2 -21264.074} C_VEL
LIN {X 0,Y 206.74,Z 549.542,A -85,B 0,C 180,E1 -21268.419,E2 -21268.419} C_VEL
LIN {X 0,Y 206.698,Z 549.55,A -85,B 0,C 180,E1 -21272.957,E2 -21272.957} C_VEL
LIN {X 0,Y 206.675,Z 549.55,A -85,B 0,C 180,E1 -21277.74,E2 -21277.74} C_VEL
LIN {X 0,Y 206.639,Z 549.556,A -85,B 0,C 180,E1 -21281.563,E2 -21281.563} C_VEL
LIN {X 0,Y 206.632,Z 549.557,A -85,B 0,C 180,E1 -21285.581,E2 -21285.581} C_VEL
LIN {X 0,Y 206.824,Z 549.534,A -85,B 0,C 180,E1 -21291.402,E2 -21291.402} C_VEL
LIN {X 0,Y 207.009,Z 549.717,A -85,B 0,C 180,E1 -21293.419,E2 -21293.419} C_VEL
LIN {X 0,Y 209.253,Z 560.547,A -85,B 0,C 180,E1 -21298.629,E2 -21298.629} C_VEL
LIN {X 0,Y 209.628,Z 563.096,A -85,B 0,C 180,E1 -21299.809,E2 -21299.809} C_VEL
LIN {X 0,Y 207.92,Z 572.738,A -85,B 0,C 180,E1 -21304.135,E2 -21304.135} C_VEL
LIN {X 0,Y 207.966,Z 581.784,A -85,B 0,C 180,E1 -21304.709,E2 -21304.709} C_VEL
LIN {X 0,Y 208.984,Z 609.406,A -85,B 0,C 180,E1 -21306.27,E2 -21306.27} C_VEL
LIN {X 0,Y 208.504,Z 615.211,A -85,B 0,C 180,E1 -21306.563,E2 -21306.563} C_VEL
LIN {X 0,Y 203.92,Z 634.253,A -85,B 0,C 180,E1 -21307.443,E2 -21307.443} C_VEL
LIN {X 0,Y 203.714,Z 640.034,A -85,B 0,C 180,E1 -21307.765,E2 -21307.765} C_VEL
LIN {X 0,Y 204.592,Z 656.573,A -85,B 0,C 180,E1 -21308.761,E2 -21308.761} C_VEL
LIN {X 0,Y 203.878,Z 669.661,A -85,B 0,C 180,E1 -21309.836,E2 -21309.836} C_VEL
LIN {X 0,Y 203.102,Z 680.365,A -85,B 0,C 180,E1 -21311.071,E2 -21311.071} C_VEL
LIN {X 0,Y 201.909,Z 691.679,A -85,B 0,C 180,E1 -21312.791,E2 -21312.791} C_VEL
LIN {X 0,Y 200.701,Z 702.9,A -85,B 0,C 180,E1 -21315.034,E2 -21315.034} C_VEL
LIN {X 0,Y 199.994,Z 711.81,A -85,B 0,C 180,E1 -21317.313,E2 -21317.313} C_VEL
LIN {X 0,Y 199.448,Z 719.746,A -85,B 0,C 180,E1 -21319.852,E2 -21319.852} C_VEL
LIN {X 0,Y 199.423,Z 727.196,A -85,B 0,C 180,E1 -21322.915,E2 -21322.915} C_VEL
LIN {X 0,Y 199.878,Z 732.815,A -85,B 0,C 180,E1 -21325.967,E2 -21325.967} C_VEL
LIN {X 0,Y 200.262,Z 735.666,A -85,B 0,C 180,E1 -21327.989,E2 -21327.989} C_VEL
LIN {X 0,Y 200.582,Z 737.787,A -85,B 0,C 180,E1 -21330,E2 -21330} C_VEL
LIN {X 0,Y 199.848,Z 739.099,A -85,B 0,C 180,E1 -21332.015,E2 -21332.015} C_VEL
LIN {X 0,Y 199.127,Z 739.825,A -85,B 0,C 180,E1 -21334.048,E2 -21334.048} C_VEL
LIN {X 0,Y 198.447,Z 740.036,A -85,B 0,C 180,E1 -21337.428,E2 -21337.428} C_VEL
LIN {X 0,Y 198.393,Z 739.26,A -85,B 0,C 180,E1 -21340.202,E2 -21340.202} C_VEL
LIN {X 0,Y 198.725,Z 738.183,A -85,B 0,C 180,E1 -21342.25,E2 -21342.25} C_VEL
LIN {X 0,Y 199.354,Z 736.623,A -85,B 0,C 180,E1 -21344.286,E2 -21344.286} C_VEL
LIN {X 0,Y 201.15,Z 733.459,A -85,B 0,C 180,E1 -21347.276,E2 -21347.276} C_VEL
LIN {X 0,Y 203.614,Z 729.176,A -85,B 0,C 180,E1 -21350.191,E2 -21350.191} C_VEL
LIN {X 0,Y 207.453,Z 722.651,A -85,B 0,C 180,E1 -21353.456,E2 -21353.456} C_VEL
LIN {X 0,Y 211.528,Z 715.508,A -85,B 0,C 180,E1 -21356.118,E2 -21356.118} C_VEL
LIN {X 0,Y 216.261,Z 706.579,A -85,B 0,C 180,E1 -21358.642,E2 -21358.642} C_VEL
LIN {X 0,Y 220.627,Z 697.544,A -85,B 0,C 180,E1 -21360.641,E2 -21360.641} C_VEL
LIN {X 0,Y 225.623,Z 685.982,A -85,B 0,C 180,E1 -21362.574,E2 -21362.574} C_VEL
LIN {X 0,Y 229.726,Z 675.085,A -85,B 0,C 180,E1 -21363.931,E2 -21363.931} C_VEL
LIN {X 0,Y 233.437,Z 663.108,A -85,B 0,C 180,E1 -21365.11,E2 -21365.11} C_VEL
LIN {X 0,Y 236.199,Z 648.646,A -85,B 0,C 180,E1 -21366.393,E2 -21366.393} C_VEL
LIN {X 0,Y 237.126,Z 636.786,A -85,B 0,C 180,E1 -21367.407,E2 -21367.407} C_VEL
LIN {X 0,Y 237.067,Z 622.667,A -85,B 0,C 180,E1 -21368.766,E2 -21368.766} C_VEL
LIN {X 0,Y 236.457,Z 607.915,A -85,B 0,C 180,E1 -21370.558,E2 -21370.558} C_VEL
LIN {X 0,Y 236.123,Z 604.65,A -85,B 0,C 180,E1 -21371.072,E2 -21371.072} C_VEL
LIN {X 0,Y 234.09,Z 596.526,A -85,B 0,C 180,E1 -21373.228,E2 -21373.228} C_VEL
LIN {X 0,Y 232.05,Z 589.347,A -85,B 0,C 180,E1 -21375.703,E2 -21375.703} C_VEL
LIN {X 0,Y 230.849,Z 586.349,A -85,B 0,C 180,E1 -21377.239,E2 -21377.239} C_VEL
LIN {X 0,Y 230.417,Z 585.527,A -85,B 0,C 180,E1 -21377.854,E2 -21377.854} C_VEL
LIN {X 0,Y 228.375,Z 582.917,A -85,B 0,C 180,E1 -21381.349,E2 -21381.349} C_VEL
LIN {X 0,Y 227.888,Z 581.213,A -85,B 0,C 180,E1 -21383.303,E2 -21383.303} C_VEL
LIN {X 0,Y 227.825,Z 581.086,A -85,B 0,C 180,E1 -21387.545,E2 -21387.545} C_VEL
LIN {X 0,Y 228.069,Z 581.815,A -85,B 0,C 180,E1 -21388.831,E2 -21388.831} C_VEL
LIN {X 0,Y 229.957,Z 585.081,A -85,B 0,C 180,E1 -21392.873,E2 -21392.873} C_VEL
LIN {X 0,Y 230.913,Z 585.987,A -85,B 0,C 180,E1 -21394.009,E2 -21394.009} C_VEL
LIN {X 0,Y 232.977,Z 589.447,A -85,B 0,C 180,E1 -21396.304,E2 -21396.304} C_VEL
LIN {X 0,Y 233.814,Z 590.531,A -85,B 0,C 180,E1 -21397.037,E2 -21397.037} C_VEL
LIN {X 0,Y 236.736,Z 595.272,A -85,B 0,C 180,E1 -21399.371,E2 -21399.371} C_VEL
LIN {X 0,Y 239.706,Z 600.549,A -85,B 0,C 180,E1 -21401.408,E2 -21401.408} C_VEL
LIN {X 0,Y 242.857,Z 607.085,A -85,B 0,C 180,E1 -21403.449,E2 -21403.449} C_VEL
LIN {X 0,Y 240.963,Z 619.662,A -85,B 0,C 180,E1 -21404.532,E2 -21404.532} C_VEL
LIN {X 0,Y 238.58,Z 630.53,A -85,B 0,C 180,E1 -21405.717,E2 -21405.717} C_VEL
LIN {X 0,Y 235.347,Z 641.608,A -85,B 0,C 180,E1 -21407.278,E2 -21407.278} C_VEL
LIN {X 0,Y 231.751,Z 651.526,A -85,B 0,C 180,E1 -21409.075,E2 -21409.075} C_VEL
LIN {X 0,Y 227.538,Z 660.914,A -85,B 0,C 180,E1 -21411.251,E2 -21411.251} C_VEL
LIN {X 0,Y 223.306,Z 668.985,A -85,B 0,C 180,E1 -21413.676,E2 -21413.676} C_VEL
LIN {X 0,Y 219.129,Z 675.712,A -85,B 0,C 180,E1 -21416.323,E2 -21416.323} C_VEL
LIN {X 0,Y 214.901,Z 681.338,A -85,B 0,C 180,E1 -21419.352,E2 -21419.352} C_VEL
LIN {X 0,Y 211.053,Z 685.558,A -85,B 0,C 180,E1 -21422.607,E2 -21422.607} C_VEL
LIN {X 0,Y 207.879,Z 688.126,A -85,B 0,C 180,E1 -21425.822,E2 -21425.822} C_VEL
LIN {X 0,Y 205.908,Z 689.188,A -85,B 0,C 180,E1 -21428.193,E2 -21428.193} C_VEL
LIN {X 0,Y 203.378,Z 689.478,A -85,B 0,C 180,E1 -21431.967,E2 -21431.967} C_VEL
LIN {X 0,Y 202.292,Z 688.978,A -85,B 0,C 180,E1 -21434.076,E2 -21434.076} C_VEL
LIN {X 0,Y 201.407,Z 687.952,A -85,B 0,C 180,E1 -21436.211,E2 -21436.211} C_VEL
LIN {X 0,Y 200.593,Z 685.971,A -85,B 0,C 180,E1 -21438.924,E2 -21438.924} C_VEL
LIN {X 0,Y 200.016,Z 681.831,A -85,B 0,C 180,E1 -21442.738,E2 -21442.738} C_VEL
LIN {X 0,Y 200.029,Z 676.778,A -85,B 0,C 180,E1 -21446.053,E2 -21446.053} C_VEL
LIN {X 0,Y 200.484,Z 670.195,A -85,B 0,C 180,E1 -21449.392,E2 -21449.392} C_VEL
LIN {X 0,Y 201.188,Z 662.693,A -85,B 0,C 180,E1 -21452.376,E2 -21452.376} C_VEL
LIN {X 0,Y 202.044,Z 654.448,A -85,B 0,C 180,E1 -21455.027,E2 -21455.027} C_VEL
LIN {X 0,Y 203.221,Z 644.185,A -85,B 0,C 180,E1 -21457.683,E2 -21457.683} C_VEL
LIN {X 0,Y 204.334,Z 633.797,A -85,B 0,C 180,E1 -21459.838,E2 -21459.838} C_VEL
LIN {X 0,Y 205.359,Z 623.322,A -85,B 0,C 180,E1 -21461.588,E2 -21461.588} C_VEL
LIN {X 0,Y 206.381,Z 610.48,A -85,B 0,C 180,E1 -21463.25,E2 -21463.25} C_VEL
LIN {X 0,Y 207.14,Z 597.572,A -85,B 0,C 180,E1 -21464.476,E2 -21464.476} C_VEL
LIN {X 0,Y 207.564,Z 583.542,A -85,B 0,C 180,E1 -21465.373,E2 -21465.373} C_VEL
LIN {X 0,Y 207.441,Z 576.034,A -85,B 0,C 180,E1 -21465.757,E2 -21465.757} C_VEL
LIN {X 0,Y 199.999,Z 551.579,A -85,B 0,C 180,E1 -21467.477,E2 -21467.477} C_VEL
LIN {X 0,Y 199.791,Z 550.57,A -85,B 0,C 180,E1 -21467.809,E2 -21467.809} C_VEL
LIN {X 0,Y 199.654,Z 550.429,A -85,B 0,C 180,E1 -21473.245,E2 -21473.245} C_VEL
LIN {X 0,Y 199.706,Z 550.42,A -85,B 0,C 180,E1 -21478.139,E2 -21478.139} C_VEL
LIN {X 0,Y 199.689,Z 550.421,A -85,B 0,C 180,E1 -21482.773,E2 -21482.773} C_VEL
LIN {X 0,Y 199.74,Z 550.415,A -85,B 0,C 180,E1 -21487.23,E2 -21487.23} C_VEL
LIN {X 0,Y 199.798,Z 550.408,A -85,B 0,C 180,E1 -21491.76,E2 -21491.76} C_VEL
LIN {X 0,Y 199.825,Z 550.407,A -85,B 0,C 180,E1 -21495.748,E2 -21495.748} C_VEL
LIN {X 0,Y 200.026,Z 550.38,A -85,B 0,C 180,E1 -21499.882,E2 -21499.882} C_VEL
LIN {X 0,Y 200.019,Z 550.381,A -85,B 0,C 180,E1 -21503.949,E2 -21503.949} C_VEL
LIN {X 0,Y 200.323,Z 550.344,A -85,B 0,C 180,E1 -21507.99,E2 -21507.99} C_VEL
LIN {X 0,Y 200.484,Z 550.321,A -85,B 0,C 180,E1 -21510,E2 -21510} C_VEL
LIN {X 0,Y 200.026,Z 550.381,A -85,B 0,C 180,E1 -21514.03,E2 -21514.03} C_VEL
LIN {X 0,Y 200.086,Z 550.372,A -85,B 0,C 180,E1 -21518.077,E2 -21518.077} C_VEL
LIN {X 0,Y 199.879,Z 550.399,A -85,B 0,C 180,E1 -21522.179,E2 -21522.179} C_VEL
LIN {X 0,Y 199.809,Z 550.407,A -85,B 0,C 180,E1 -21526.343,E2 -21526.343} C_VEL
LIN {X 0,Y 199.695,Z 550.419,A -85,B 0,C 180,E1 -21530.606,E2 -21530.606} C_VEL
LIN {X 0,Y 199.668,Z 550.424,A -85,B 0,C 180,E1 -21534.985,E2 -21534.985} C_VEL
LIN {X 0,Y 199.667,Z 550.422,A -85,B 0,C 180,E1 -21539.523,E2 -21539.523} C_VEL
LIN {X 0,Y 199.66,Z 550.427,A -85,B 0,C 180,E1 -21542.349,E2 -21542.349} C_VEL
LIN {X 0,Y 199.655,Z 550.421,A -85,B 0,C 180,E1 -21546.755,E2 -21546.755} C_VEL
LIN {X 0,Y 199.68,Z 550.422,A -85,B 0,C 180,E1 -21549.31,E2 -21549.31} C_VEL
LIN {X 0,Y 199.664,Z 550.426,A -85,B 0,C 180,E1 -21552.337,E2 -21552.337} C_VEL
LIN {X 0,Y 199.632,Z 550.425,A -85,B 0,C 180,E1 -21555.242,E2 -21555.242} C_VEL
LIN {X 0,Y 199.641,Z 550.428,A -85,B 0,C 180,E1 -21560.755,E2 -21560.755} C_VEL
LIN {X 0,Y 199.634,Z 550.425,A -85,B 0,C 180,E1 -21565.717,E2 -21565.717} C_VEL
LIN {X 0,Y 199.703,Z 550.422,A -85,B 0,C 180,E1 -21568.136,E2 -21568.136} C_VEL
LIN {X 0,Y 199.686,Z 550.419,A -85,B 0,C 180,E1 -21572.771,E2 -21572.771} C_VEL
LIN {X 0,Y 199.748,Z 550.414,A -85,B 0,C 180,E1 -21577.229,E2 -21577.229} C_VEL
LIN {X 0,Y 199.836,Z 550.401,A -85,B 0,C 180,E1 -21581.721,E2 -21581.721} C_VEL
LIN {X 0,Y 199.833,Z 550.404,A -85,B 0,C 180,E1 -21585.747,E2 -21585.747} C_VEL
LIN {X 0,Y 200.068,Z 550.374,A -85,B 0,C 180,E1 -21589.883,E2 -21589.883} C_VEL
LIN {X 0,Y 200.035,Z 550.378,A -85,B 0,C 180,E1 -21593.949,E2 -21593.949} C_VEL
LIN {X 0,Y 200.318,Z 550.344,A -85,B 0,C 180,E1 -21597.989,E2 -21597.989} C_VEL
LIN {X 0,Y 200.475,Z 550.321,A -85,B 0,C 180,E1 -21599.999,E2 -21599.999} C_VEL
LIN {X 0,Y 200.026,Z 550.38,A -85,B 0,C 180,E1 -21604.029,E2 -21604.029} C_VEL
LIN {X 0,Y 200.106,Z 550.369,A -85,B 0,C 180,E1 -21608.075,E2 -21608.075} C_VEL
LIN {X 0,Y 199.909,Z 550.394,A -85,B 0,C 180,E1 -21612.176,E2 -21612.176} C_VEL
LIN {X 0,Y 199.799,Z 550.409,A -85,B 0,C 180,E1 -21616.343,E2 -21616.343} C_VEL
LIN {X 0,Y 199.677,Z 550.424,A -85,B 0,C 180,E1 -21620.607,E2 -21620.607} C_VEL
LIN {X 0,Y 199.661,Z 550.425,A -85,B 0,C 180,E1 -21624.985,E2 -21624.985} C_VEL
LIN {X 0,Y 199.671,Z 550.423,A -85,B 0,C 180,E1 -21629.522,E2 -21629.522} C_VEL
LIN {X 0,Y 199.674,Z 550.425,A -85,B 0,C 180,E1 -21632.358,E2 -21632.358} C_VEL
LIN {X 0,Y 199.619,Z 550.429,A -85,B 0,C 180,E1 -21636.763,E2 -21636.763} C_VEL
LIN {X 0,Y 199.605,Z 550.433,A -85,B 0,C 180,E1 -21639.328,E2 -21639.328} C_VEL
LIN {X 0,Y 199.571,Z 550.437,A -85,B 0,C 180,E1 -21642.31,E2 -21642.31} C_VEL
LIN {X 0,Y 199.579,Z 550.437,A -85,B 0,C 180,E1 -21645.229,E2 -21645.229} C_VEL
LIN {X 0,Y 199.724,Z 550.42,A -85,B 0,C 180,E1 -21650.727,E2 -21650.727} C_VEL
LIN {X 0,Y 199.984,Z 550.534,A -85,B 0,C 180,E1 -21653.488,E2 -21653.488} C_VEL
LIN {X 0,Y 202.339,Z 561.708,A -85,B 0,C 180,E1 -21659.073,E2 -21659.073} C_VEL
LIN {X 0,Y 202.339,Z 564.197,A -85,B 0,C 180,E1 -21660.266,E2 -21660.266} C_VEL
LIN {X 0,Y 200.998,Z 571.327,A -85,B 0,C 180,E1 -21663.596,E2 -21663.596} C_VEL
LIN {X 0,Y 200.927,Z 575.545,A -85,B 0,C 180,E1 -21663.935,E2 -21663.935} C_VEL
LIN {X 0,Y 202.202,Z 613.822,A -85,B 0,C 180,E1 -21666.203,E2 -21666.203} C_VEL
LIN {X 0,Y 203.714,Z 640.034,A -85,B 0,C 180,E1 -21667.765,E2 -21667.765} C_VEL
LIN {X 0,Y 203.428,Z 645.829,A -85,B 0,C 180,E1 -21668.081,E2 -21668.081} C_VEL
LIN {X 0,Y 200.824,Z 655.267,A -85,B 0,C 180,E1 -21668.566,E2 -21668.566} C_VEL
LIN {X 0,Y 197.767,Z 664.558,A -85,B 0,C 180,E1 -21669.211,E2 -21669.211} C_VEL
LIN {X 0,Y 196.757,Z 670.145,A -85,B 0,C 180,E1 -21669.761,E2 -21669.761} C_VEL
LIN {X 0,Y 195.914,Z 681.306,A -85,B 0,C 180,E1 -21671.165,E2 -21671.165} C_VEL
LIN {X 0,Y 194.71,Z 692.113,A -85,B 0,C 180,E1 -21672.946,E2 -21672.946} C_VEL
LIN {X 0,Y 193.667,Z 701.942,A -85,B 0,C 180,E1 -21675.016,E2 -21675.016} C_VEL
LIN {X 0,Y 192.964,Z 710.823,A -85,B 0,C 180,E1 -21677.378,E2 -21677.378} C_VEL
LIN {X 0,Y 192.456,Z 718.622,A -85,B 0,C 180,E1 -21679.966,E2 -21679.966} C_VEL
LIN {X 0,Y 192.418,Z 725.057,A -85,B 0,C 180,E1 -21682.655,E2 -21682.655} C_VEL
LIN {X 0,Y 192.864,Z 730.945,A -85,B 0,C 180,E1 -21685.821,E2 -21685.821} C_VEL
LIN {X 0,Y 193.443,Z 735.12,A -85,B 0,C 180,E1 -21688.959,E2 -21688.959} C_VEL
LIN {X 0,Y 193.626,Z 736.188,A -85,B 0,C 180,E1 -21690,E2 -21690} C_VEL
LIN {X 0,Y 192.871,Z 737.587,A -85,B 0,C 180,E1 -21692.088,E2 -21692.088} C_VEL
LIN {X 0,Y 192.102,Z 738.466,A -85,B 0,C 180,E1 -21694.196,E2 -21694.196} C_VEL
LIN {X 0,Y 191.443,Z 738.86,A -85,B 0,C 180,E1 -21697.617,E2 -21697.617} C_VEL
LIN {X 0,Y 191.393,Z 738.254,A -85,B 0,C 180,E1 -21700.579,E2 -21700.579} C_VEL
LIN {X 0,Y 191.778,Z 737.284,A -85,B 0,C 180,E1 -21702.701,E2 -21702.701} C_VEL
LIN {X 0,Y 192.461,Z 735.893,A -85,B 0,C 180,E1 -21704.81,E2 -21704.81} C_VEL
LIN {X 0,Y 194.368,Z 732.964,A -85,B 0,C 180,E1 -21707.899,E2 -21707.899} C_VEL
LIN {X 0,Y 196.967,Z 728.953,A -85,B 0,C 180,E1 -21710.904,E2 -21710.904} C_VEL
LIN {X 0,Y 200.959,Z 722.768,A -85,B 0,C 180,E1 -21714.262,E2 -21714.262} C_VEL
LIN {X 0,Y 205.212,Z 716.004,A -85,B 0,C 180,E1 -21716.986,E2 -21716.986} C_VEL
LIN {X 0,Y 210.101,Z 707.631,A -85,B 0,C 180,E1 -21719.563,E2 -21719.563} C_VEL
LIN {X 0,Y 214.611,Z 699.051,A -85,B 0,C 180,E1 -21721.597,E2 -21721.597} C_VEL
LIN {X 0,Y 219.744,Z 688.334,A -85,B 0,C 180,E1 -21723.553,E2 -21723.553} C_VEL
LIN {X 0,Y 224.545,Z 676.929,A -85,B 0,C 180,E1 -21725.107,E2 -21725.107} C_VEL
LIN {X 0,Y 228.613,Z 665.135,A -85,B 0,C 180,E1 -21726.347,E2 -21726.347} C_VEL
LIN {X 0,Y 231.563,Z 652.573,A -85,B 0,C 180,E1 -21727.526,E2 -21727.526} C_VEL
LIN {X 0,Y 233.216,Z 640.115,A -85,B 0,C 180,E1 -21728.649,E2 -21728.649} C_VEL
LIN {X 0,Y 233.585,Z 627.773,A -85,B 0,C 180,E1 -21729.869,E2 -21729.869} C_VEL
LIN {X 0,Y 233.331,Z 613.738,A -85,B 0,C 180,E1 -21731.532,E2 -21731.532} C_VEL
LIN {X 0,Y 233.113,Z 609.034,A -85,B 0,C 180,E1 -21732.233,E2 -21732.233} C_VEL
LIN {X 0,Y 231.307,Z 601.356,A -85,B 0,C 180,E1 -21734.381,E2 -21734.381} C_VEL
LIN {X 0,Y 229.822,Z 595.023,A -85,B 0,C 180,E1 -21736.61,E2 -21736.61} C_VEL
LIN {X 0,Y 228.915,Z 592.523,A -85,B 0,C 180,E1 -21737.988,E2 -21737.988} C_VEL
LIN {X 0,Y 226.886,Z 589.68,A -85,B 0,C 180,E1 -21741.72,E2 -21741.72} C_VEL
LIN {X 0,Y 226.44,Z 588.062,A -85,B 0,C 180,E1 -21743.865,E2 -21743.865} C_VEL
LIN {X 0,Y 226.514,Z 588.109,A -85,B 0,C 180,E1 -21747.678,E2 -21747.678} C_VEL
LIN {X 0,Y 228.447,Z 591.974,A -85,B 0,C 180,E1 -21752.679,E2 -21752.679} C_VEL
LIN {X 0,Y 229.19,Z 592.749,A -85,B 0,C 180,E1 -21753.606,E2 -21753.606} C_VEL
LIN {X 0,Y 231.481,Z 596.48,A -85,B 0,C 180,E1 -21756.216,E2 -21756.216} C_VEL
LIN {X 0,Y 234.483,Z 601.636,A -85,B 0,C 180,E1 -21758.835,E2 -21758.835} C_VEL
LIN {X 0,Y 237.381,Z 607.445,A -85,B 0,C 180,E1 -21761.065,E2 -21761.065} C_VEL
LIN {X 0,Y 238.872,Z 611.018,A -85,B 0,C 180,E1 -21762.25,E2 -21762.25} C_VEL
LIN {X 0,Y 236.82,Z 622.866,A -85,B 0,C 180,E1 -21763.31,E2 -21763.31} C_VEL
LIN {X 0,Y 234.173,Z 633.459,A -85,B 0,C 180,E1 -21764.53,E2 -21764.53} C_VEL
LIN {X 0,Y 230.679,Z 644.273,A -85,B 0,C 180,E1 -21766.119,E2 -21766.119} C_VEL
LIN {X 0,Y 226.879,Z 653.886,A -85,B 0,C 180,E1 -21767.931,E2 -21767.931} C_VEL
LIN {X 0,Y 222.738,Z 662.557,A -85,B 0,C 180,E1 -21769.979,E2 -21769.979} C_VEL
LIN {X 0,Y 218.848,Z 669.55,A -85,B 0,C 180,E1 -21772.11,E2 -21772.11} C_VEL
LIN {X 0,Y 214.924,Z 675.473,A -85,B 0,C 180,E1 -21774.371,E2 -21774.371} C_VEL
LIN {X 0,Y 210.616,Z 681.136,A -85,B 0,C 180,E1 -21777.192,E2 -21777.192} C_VEL
LIN {X 0,Y 206.881,Z 685.231,A -85,B 0,C 180,E1 -21780.001,E2 -21780.001} C_VEL
LIN {X 0,Y 204.004,Z 687.795,A -85,B 0,C 180,E1 -21782.524,E2 -21782.524} C_VEL
LIN {X 0,Y 200.554,Z 689.988,A -85,B 0,C 180,E1 -21786.035,E2 -21786.035} C_VEL
LIN {X 0,Y 198.802,Z 690.622,A -85,B 0,C 180,E1 -21788.182,E2 -21788.182} C_VEL
LIN {X 0,Y 197.325,Z 690.762,A -85,B 0,C 180,E1 -21790.259,E2 -21790.259} C_VEL
LIN {X 0,Y 195.352,Z 689.955,A -85,B 0,C 180,E1 -21793.753,E2 -21793.753} C_VEL
LIN {X 0,Y 194.124,Z 688.24,A -85,B 0,C 180,E1 -21796.837,E2 -21796.837} C_VEL
LIN {X 0,Y 193.25,Z 685.285,A -85,B 0,C 180,E1 -21800.212,E2 -21800.212} C_VEL
LIN {X 0,Y 192.884,Z 681.069,A -85,B 0,C 180,E1 -21803.629,E2 -21803.629} C_VEL
LIN {X 0,Y 193.056,Z 675.387,A -85,B 0,C 180,E1 -21807.069,E2 -21807.069} C_VEL
LIN {X 0,Y 193.593,Z 668.027,A -85,B 0,C 180,E1 -21810.548,E2 -21810.548} C_VEL
LIN {X 0,Y 194.534,Z 659.193,A -85,B 0,C 180,E1 -21813.808,E2 -21813.808} C_VEL
LIN {X 0,Y 195.473,Z 650.551,A -85,B 0,C 180,E1 -21816.388,E2 -21816.388} C_VEL
LIN {X 0,Y 196.654,Z 640.202,A -85,B 0,C 180,E1 -21818.875,E2 -21818.875} C_VEL
LIN {X 0,Y 197.873,Z 628.708,A -85,B 0,C 180,E1 -21821.079,E2 -21821.079} C_VEL
LIN {X 0,Y 199.023,Z 615.665,A -85,B 0,C 180,E1 -21822.999,E2 -21822.999} C_VEL
LIN {X 0,Y 199.863,Z 603.433,A -85,B 0,C 180,E1 -21824.339,E2 -21824.339} C_VEL
LIN {X 0,Y 200.434,Z 590.359,A -85,B 0,C 180,E1 -21825.364,E2 -21825.364} C_VEL
LIN {X 0,Y 200.547,Z 577.489,A -85,B 0,C 180,E1 -21826.06,E2 -21826.06} C_VEL
LIN {X 0,Y 192.925,Z 552.326,A -85,B 0,C 180,E1 -21827.894,E2 -21827.894} C_VEL
LIN {X 0,Y 192.687,Z 551.41,A -85,B 0,C 180,E1 -21828.27,E2 -21828.27} C_VEL
LIN {X 0,Y 192.62,Z 551.305,A -85,B 0,C 180,E1 -21833.39,E2 -21833.39} C_VEL
LIN {X 0,Y 192.61,Z 551.306,A -85,B 0,C 180,E1 -21837.061,E2 -21837.061} C_VEL
LIN {X 0,Y 192.667,Z 551.298,A -85,B 0,C 180,E1 -21841.693,E2 -21841.693} C_VEL
LIN {X 0,Y 192.709,Z 551.29,A -85,B 0,C 180,E1 -21846.35,E2 -21846.35} C_VEL
LIN {X 0,Y 192.733,Z 551.29,A -85,B 0,C 180,E1 -21851.46,E2 -21851.46} C_VEL
LIN {X 0,Y 192.753,Z 551.284,A -85,B 0,C 180,E1 -21855.213,E2 -21855.213} C_VEL
LIN {X 0,Y 192.949,Z 551.264,A -85,B 0,C 180,E1 -21859.567,E2 -21859.567} C_VEL
LIN {X 0,Y 192.982,Z 551.256,A -85,B 0,C 180,E1 -21863.728,E2 -21863.728} C_VEL
LIN {X 0,Y 193.265,Z 551.223,A -85,B 0,C 180,E1 -21867.916,E2 -21867.916} C_VEL
LIN {X 0,Y 193.448,Z 551.197,A -85,B 0,C 180,E1 -21870,E2 -21870} C_VEL
LIN {X 0,Y 192.972,Z 551.259,A -85,B 0,C 180,E1 -21874.177,E2 -21874.177} C_VEL
LIN {X 0,Y 193.035,Z 551.249,A -85,B 0,C 180,E1 -21878.374,E2 -21878.374} C_VEL
LIN {X 0,Y 192.806,Z 551.278,A -85,B 0,C 180,E1 -21882.633,E2 -21882.633} C_VEL
LIN {X 0,Y 192.762,Z 551.283,A -85,B 0,C 180,E1 -21886.958,E2 -21886.958} C_VEL
LIN {X 0,Y 192.626,Z 551.3,A -85,B 0,C 180,E1 -21891.398,E2 -21891.398} C_VEL
LIN {X 0,Y 192.65,Z 551.3,A -85,B 0,C 180,E1 -21894.213,E2 -21894.213} C_VEL
LIN {X 0,Y 192.647,Z 551.296,A -85,B 0,C 180,E1 -21898.888,E2 -21898.888} C_VEL
LIN {X 0,Y 192.6,Z 551.305,A -85,B 0,C 180,E1 -21903.185,E2 -21903.185} C_VEL
LIN {X 0,Y 192.602,Z 551.305,A -85,B 0,C 180,E1 -21908.339,E2 -21908.339} C_VEL
LIN {X 0,Y 192.601,Z 551.304,A -85,B 0,C 180,E1 -21913.129,E2 -21913.129} C_VEL
LIN {X 0,Y 192.538,Z 551.31,A -85,B 0,C 180,E1 -21916.888,E2 -21916.888} C_VEL
LIN {X 0,Y 192.574,Z 551.309,A -85,B 0,C 180,E1 -21921.652,E2 -21921.652} C_VEL
LIN {X 0,Y 192.598,Z 551.303,A -85,B 0,C 180,E1 -21924.277,E2 -21924.277} C_VEL
LIN {X 0,Y 192.606,Z 551.304,A -85,B 0,C 180,E1 -21929.279,E2 -21929.279} C_VEL
LIN {X 0,Y 192.664,Z 551.296,A -85,B 0,C 180,E1 -21931.691,E2 -21931.691} C_VEL
LIN {X 0,Y 192.71,Z 551.293,A -85,B 0,C 180,E1 -21936.348,E2 -21936.348} C_VEL
LIN {X 0,Y 192.78,Z 551.28,A -85,B 0,C 180,E1 -21941.412,E2 -21941.412} C_VEL
LIN {X 0,Y 192.761,Z 551.284,A -85,B 0,C 180,E1 -21945.213,E2 -21945.213} C_VEL
LIN {X 0,Y 192.979,Z 551.256,A -85,B 0,C 180,E1 -21949.508,E2 -21949.508} C_VEL
LIN {X 0,Y 193.065,Z 551.242,A -85,B 0,C 180,E1 -21951.627,E2 -21951.627} C_VEL
LIN {X 0,Y 193.26,Z 551.223,A -85,B 0,C 180,E1 -21957.915,E2 -21957.915} C_VEL
LIN {X 0,Y 193.439,Z 551.198,A -85,B 0,C 180,E1 -21959.999,E2 -21959.999} C_VEL
LIN {X 0,Y 192.973,Z 551.259,A -85,B 0,C 180,E1 -21964.176,E2 -21964.176} C_VEL
LIN {X 0,Y 193.057,Z 551.247,A -85,B 0,C 180,E1 -21968.372,E2 -21968.372} C_VEL
LIN {X 0,Y 192.848,Z 551.277,A -85,B 0,C 180,E1 -21972.63,E2 -21972.63} C_VEL
LIN {X 0,Y 192.753,Z 551.283,A -85,B 0,C 180,E1 -21976.958,E2 -21976.958} C_VEL
LIN {X 0,Y 192.612,Z 551.303,A -85,B 0,C 180,E1 -21981.399,E2 -21981.399} C_VEL
LIN {X 0,Y 192.643,Z 551.3,A -85,B 0,C 180,E1 -21984.213,E2 -21984.213} C_VEL
LIN {X 0,Y 192.646,Z 551.3,A -85,B 0,C 180,E1 -21988.892,E2 -21988.892} C_VEL
LIN {X 0,Y 192.595,Z 551.305,A -85,B 0,C 180,E1 -21993.186,E2 -21993.186} C_VEL
LIN {X 0,Y 192.548,Z 551.311,A -85,B 0,C 180,E1 -21998.352,E2 -21998.352} C_VEL
LIN {X 0,Y 192.489,Z 551.32,A -85,B 0,C 180,E1 -22003.096,E2 -22003.096} C_VEL
LIN {X 0,Y 192.516,Z 551.318,A -85,B 0,C 180,E1 -22006.896,E2 -22006.896} C_VEL
LIN {X 0,Y 192.896,Z 551.271,A -85,B 0,C 180,E1 -22013.278,E2 -22013.278} C_VEL
LIN {X 0,Y 193.018,Z 551.682,A -85,B 0,C 180,E1 -22013.838,E2 -22013.838} C_VEL
LIN {X 0,Y 195.259,Z 562.02,A -85,B 0,C 180,E1 -22019.144,E2 -22019.144} C_VEL
LIN {X 0,Y 195.171,Z 564.375,A -85,B 0,C 180,E1 -22020.322,E2 -22020.322} C_VEL
LIN {X 0,Y 194.074,Z 570.055,A -85,B 0,C 180,E1 -22023.086,E2 -22023.086} C_VEL
LIN {X 0,Y 193.985,Z 574.176,A -85,B 0,C 180,E1 -22023.436,E2 -22023.436} C_VEL
LIN {X 0,Y 195.047,Z 611.733,A -85,B 0,C 180,E1 -22025.743,E2 -22025.743} C_VEL
LIN {X 0,Y 197.536,Z 656.409,A -85,B 0,C 180,E1 -22028.542,E2 -22028.542} C_VEL
LIN {X 0,Y 196.835,Z 668.878,A -85,B 0,C 180,E1 -22029.628,E2 -22029.628} C_VEL
LIN {X 0,Y 196.757,Z 670.145,A -85,B 0,C 180,E1 -22029.761,E2 -22029.761} C_VEL
LIN {X 0,Y 196.049,Z 673.768,A -85,B 0,C 180,E1 -22030.165,E2 -22030.165} C_VEL
LIN {X 0,Y 193.372,Z 680.608,A -85,B 0,C 180,E1 -22031.05,E2 -22031.05} C_VEL
LIN {X 0,Y 188.396,Z 691.09,A -85,B 0,C 180,E1 -22032.82,E2 -22032.82} C_VEL
